FUNCTION_BLOCK "State_Machine2"   // FB71, GRAPH
VERSION : 0.1
// stored: AcknowledgeErrorsRequired true, AutoNumber false, GraphVersion 6.0, InitialValuesAcquisition false, IsIECCheckEnabled false, LanguageInNetworks LAD, LockOperatingMode false, PermanentILProcessingInMANMode false, SetENOAutomatically false, SkipSteps false, UDAEnableTagReadback false, WithAlarmHandling true
   // inherited from GRAPH_BASE
   VAR
      OFF_SQ_BASE : Bool;
   END_VAR
   VAR_INPUT
      OFF_SQ { ExternalAccessible := 'False'; ExternalVisible := 'False'; ExternalWritable := 'False'} : Bool := false;   // Disattiva catena / Turn sequence off
      INIT_SQ { ExternalAccessible := 'False'; ExternalVisible := 'False'; ExternalWritable := 'False'} : Bool := false;   // Imposta catena nello stato iniziale / Set sequence to initial state
      ACK_EF { ExternalAccessible := 'False'; ExternalVisible := 'False'; ExternalWritable := 'False'} : Bool := false;   // Conferma tutti gli errori e le anomalie / Acknowledge all errors and faults
      S_PREV { ExternalAccessible := 'False'; ExternalVisible := 'False'; ExternalWritable := 'False'} : Bool := false;   // Emetti il passo precedente nel parametro S_NO / Output previous step in parameter S_NO
      S_NEXT { ExternalAccessible := 'False'; ExternalVisible := 'False'; ExternalWritable := 'False'} : Bool := false;   // Visualizza passo successivo nel parametro S_NO / Indicate next step in parameter S_NO
      SW_AUTO { ExternalAccessible := 'False'; ExternalVisible := 'False'; ExternalWritable := 'False'} : Bool := false;   // Imposta funzionamento automatico / Automatic mode
      SW_TAP { ExternalAccessible := 'False'; ExternalVisible := 'False'; ExternalWritable := 'False'} : Bool := false;   // Semiautomatico/Avanza con transizione / Semiautomatic/switch with transition
      SW_TOP { ExternalAccessible := 'False'; ExternalVisible := 'False'; ExternalWritable := 'False'} : Bool := false;   // Semiautomatico/Ignora transizione / Semiautomatic/ignore transition
      SW_MAN { ExternalAccessible := 'False'; ExternalVisible := 'False'; ExternalWritable := 'False'} : Bool := false;   // Funzionamento manuale / Manual mode
      S_SEL { ExternalAccessible := 'False'; ExternalVisible := 'False'; ExternalWritable := 'False'} : Int := 0;   // Seleziona passo da visualizzare in S_NO / Select step to be output to S_NO
      S_ON { ExternalAccessible := 'False'; ExternalVisible := 'False'; ExternalWritable := 'False'} : Bool := false;   // Attiva passo visualizzato nel parametro S_NO / Activate step indicated in S_NO
      S_OFF { ExternalAccessible := 'False'; ExternalVisible := 'False'; ExternalWritable := 'False'} : Bool := false;   // Disattiva passo visualizzato nel parametro S_NO / Deactivate step indicated S_NO
      T_PUSH { ExternalAccessible := 'False'; ExternalVisible := 'False'; ExternalWritable := 'False'} : Bool := false;   // Abilita commutazione per la transizione nel funzionamento semiautomatico / Enable transition to switch in semi automatic mode
   END_VAR
   VAR_OUTPUT
      S_NO { ExternalAccessible := 'False'; ExternalVisible := 'False'; ExternalWritable := 'False'} : Int := 0;   // Numero del passo / Step number
      S_MORE { ExternalAccessible := 'False'; ExternalVisible := 'False'; ExternalWritable := 'False'} : Bool := false;   // Sono presenti altri passi e possono essere visualizzati in S_NO. / More steps are available and can be shown in S_NO
      S_ACTIVE { ExternalAccessible := 'False'; ExternalVisible := 'False'; ExternalWritable := 'False'} : Bool := false;   // Il passo visualizzato nel parametro S_NO è attivo / Step indicated in S_NO is active
      ERR_FLT { ExternalAccessible := 'False'; ExternalVisible := 'False'; ExternalWritable := 'False'} : Bool := false;   // Errore cumulativo interlock o supervisione / Interlock or supervision group error
      AUTO_ON { ExternalAccessible := 'False'; ExternalVisible := 'False'; ExternalWritable := 'False'} : Bool := false;   // Funzionamento automatico attivo / Automatic mode is active
      TAP_ON { ExternalAccessible := 'False'; ExternalVisible := 'False'; ExternalWritable := 'False'} : Bool := false;   // Funzionamento semiautomatico/Passo con transizione attivo / Semiautomatic mode/step with transition enabled
      TOP_ON { ExternalAccessible := 'False'; ExternalVisible := 'False'; ExternalWritable := 'False'} : Bool := false;   // Semiautomatico/Ignora transizione attivo / Semiautomatic mode/ignore transition enabled
      MAN_ON { ExternalAccessible := 'False'; ExternalVisible := 'False'; ExternalWritable := 'False'} : Bool := false;   // Funzionamento manuale attivo / Manual mode is active
   END_VAR
BEGIN
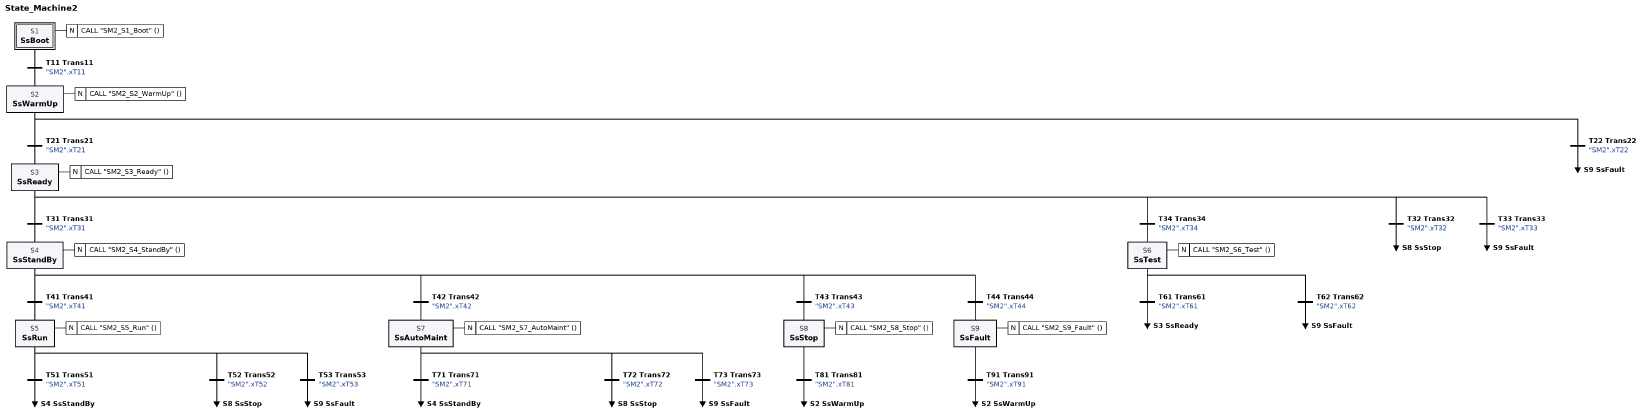
   // sequencer 1: State Machine Battery
   INITIAL_STEP SsBoot:   // S1, max time T#10S, warning time T#7S
              N    CALL "SM2_S1_Boot" ()
   END_STEP
   TRANSITION Trans11 FROM SsBoot TO SsWarmUp   // T11
      := "SM2".xT11;
   END_TRANSITION
   STEP SsWarmUp:   // S2, max time T#10S, warning time T#7S
              N    CALL "SM2_S2_WarmUp" ()
   END_STEP
   TRANSITION Trans21 FROM SsWarmUp TO SsReady   // T21
      := "SM2".xT21;
   END_TRANSITION
   TRANSITION Trans22 FROM SsWarmUp TO SsFault   // T22, jump
      := "SM2".xT22;
   END_TRANSITION
   STEP SsReady:   // S3, max time T#10S, warning time T#7S
              N    CALL "SM2_S3_Ready" ()
   END_STEP
   TRANSITION Trans31 FROM SsReady TO SsStandBy   // T31
      := "SM2".xT31;
   END_TRANSITION
   TRANSITION Trans34 FROM SsReady TO SsTest   // T34
      := "SM2".xT34;
   END_TRANSITION
   TRANSITION Trans32 FROM SsReady TO SsStop   // T32, jump
      := "SM2".xT32;
   END_TRANSITION
   TRANSITION Trans33 FROM SsReady TO SsFault   // T33, jump
      := "SM2".xT33;
   END_TRANSITION
   STEP SsStandBy:   // S4, max time T#10S, warning time T#7S
              N    CALL "SM2_S4_StandBy" ()
   END_STEP
   TRANSITION Trans41 FROM SsStandBy TO SsRun   // T41
      := "SM2".xT41;
   END_TRANSITION
   TRANSITION Trans42 FROM SsStandBy TO SsAutoMaint   // T42
      := "SM2".xT42;
   END_TRANSITION
   TRANSITION Trans43 FROM SsStandBy TO SsStop   // T43
      := "SM2".xT43;
   END_TRANSITION
   TRANSITION Trans44 FROM SsStandBy TO SsFault   // T44
      := "SM2".xT44;
   END_TRANSITION
   STEP SsRun:   // S5, max time T#10S, warning time T#7S
              N    CALL "SM2_S5_Run" ()
   END_STEP
   TRANSITION Trans51 FROM SsRun TO SsStandBy   // T51, jump
      := "SM2".xT51;
   END_TRANSITION
   TRANSITION Trans52 FROM SsRun TO SsStop   // T52, jump
      := "SM2".xT52;
   END_TRANSITION
   TRANSITION Trans53 FROM SsRun TO SsFault   // T53, jump
      := "SM2".xT53;
   END_TRANSITION
   STEP SsTest:   // S6, max time T#10S, warning time T#7S
              N    CALL "SM2_S6_Test" ()
   END_STEP
   TRANSITION Trans61 FROM SsTest TO SsReady   // T61, jump
      := "SM2".xT61;
   END_TRANSITION
   TRANSITION Trans62 FROM SsTest TO SsFault   // T62, jump
      := "SM2".xT62;
   END_TRANSITION
   STEP SsAutoMaint:   // S7, max time T#10S, warning time T#7S
              N    CALL "SM2_S7_AutoMaint" ()
   END_STEP
   TRANSITION Trans71 FROM SsAutoMaint TO SsStandBy   // T71, jump
      := "SM2".xT71;
   END_TRANSITION
   TRANSITION Trans72 FROM SsAutoMaint TO SsStop   // T72, jump
      := "SM2".xT72;
   END_TRANSITION
   TRANSITION Trans73 FROM SsAutoMaint TO SsFault   // T73, jump
      := "SM2".xT73;
   END_TRANSITION
   STEP SsStop:   // S8, max time T#10S, warning time T#7S
              N    CALL "SM2_S8_Stop" ()
   END_STEP
   TRANSITION Trans81 FROM SsStop TO SsWarmUp   // T81, jump
      := "SM2".xT81;
   END_TRANSITION
   STEP SsFault:   // S9, max time T#10S, warning time T#7S
              N    CALL "SM2_S9_Fault" ()
   END_STEP
   TRANSITION Trans91 FROM SsFault TO SsWarmUp   // T91, jump
      := "SM2".xT91;
   END_TRANSITION
END_FUNCTION_BLOCK

FUNCTION "LOGIC_PE_1" : Void   // FC7, LAD
{ S7_Optimized_Access := 'TRUE' }
VERSION : 0.1
// stored: AutoNumber true, IsIECCheckEnabled false, SetENOAutomatically false, UDAEnableTagReadback false
   VAR_TEMP
      rVac : Real;
   END_VAR
   VAR_TEMP   // added for the SCL form of the ladder/FBD networks
      _w1 : Bool;
      _w2 : Bool;
      _w3 : Bool;
   END_VAR
BEGIN

REGION Network 1: Write value of Password, P mode and Q mode - to check
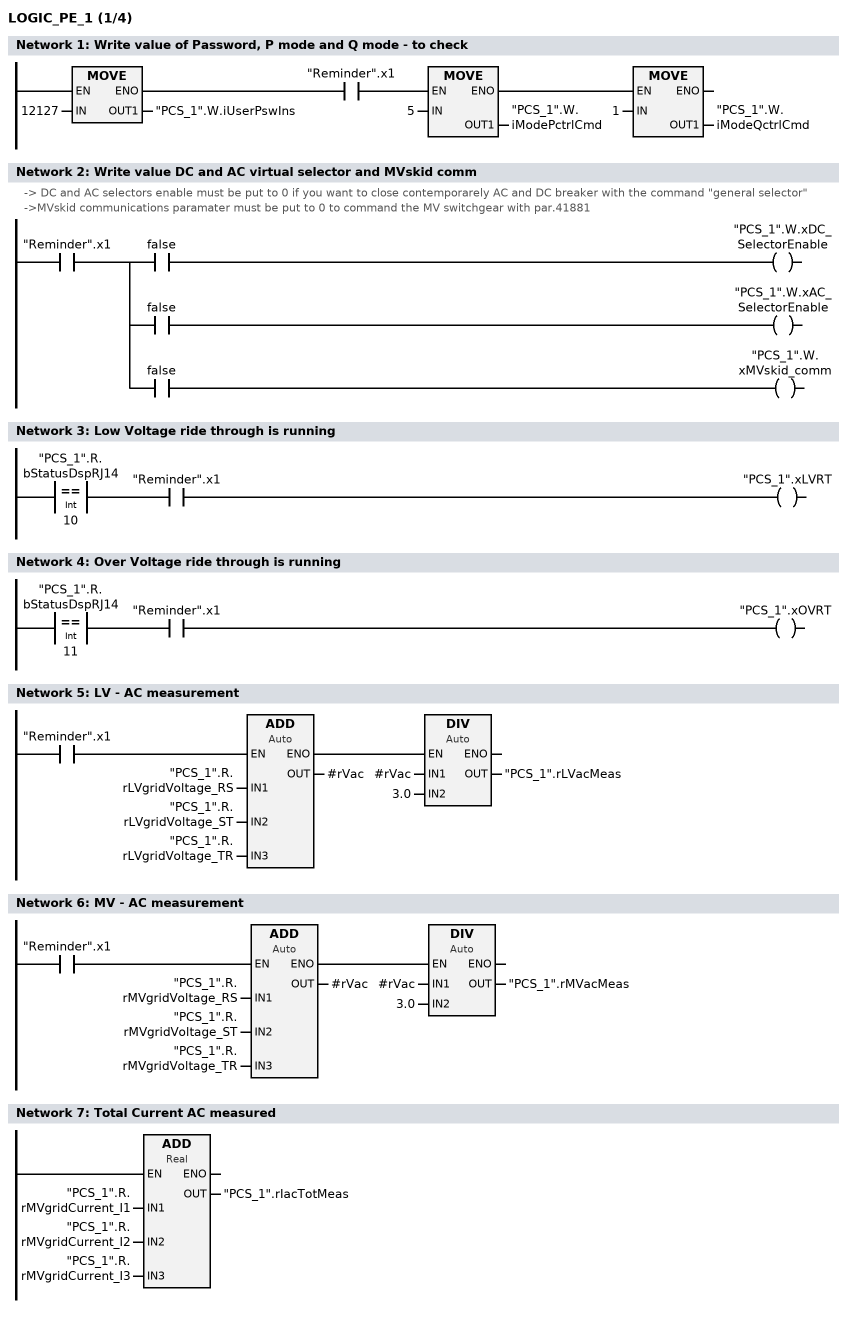
   RUNG wire#powerrail
      Move(in := 12127, out1 => "PCS_1".W.iUserPswIns)
      Contact( "Reminder".x1 )
      Move(in := 5, out1 => "PCS_1".W.iModePctrlCmd)
      Move(in := 1, out1 => "PCS_1".W.iModeQctrlCmd)
   END_RUNG
   // the same network as SCL:
   "PCS_1".W.iUserPswIns := 12127;
   IF "Reminder".x1 THEN
       "PCS_1".W.iModePctrlCmd := 5;
       "PCS_1".W.iModeQctrlCmd := 1;
   END_IF;
END_REGION

REGION Network 2: Write value DC and AC virtual selector and MVskid comm
   // -> DC and AC selectors enable must be put to 0 if you want to close contemporarely AC and DC breaker with the command "general selector"
   // ->MVskid communications paramater must be put to 0 to command the MV switchgear with par.41881
   RUNG wire#powerrail
      Contact( "Reminder".x1 )
      wire#w1
      Contact( false )
      Coil( "PCS_1".W.xDC_SelectorEnable )
   END_RUNG
   RUNG wire#w1
      Contact( false )
      Coil( "PCS_1".W.xAC_SelectorEnable )
   END_RUNG
   RUNG wire#w1
      Contact( false )
      Coil( "PCS_1".W.xMVskid_comm )
   END_RUNG
   // the same network as SCL:
   "PCS_1".W.xDC_SelectorEnable := "Reminder".x1 AND false;
   "PCS_1".W.xAC_SelectorEnable := "Reminder".x1 AND false;
   "PCS_1".W.xMVskid_comm := "Reminder".x1 AND false;
END_REGION

REGION Network 3: Low Voltage ride through is running
   RUNG wire#powerrail
      { S7_Templates := "SrcType := Int" } EQ_Contact(in1 := "PCS_1".R.bStatusDspRJ14, in2 := 10)
      Contact( "Reminder".x1 )
      Coil( "PCS_1".xLVRT )
   END_RUNG
   // the same network as SCL:
   "PCS_1".xLVRT := ("PCS_1".R.bStatusDspRJ14 = 10) AND "Reminder".x1;
END_REGION

REGION Network 4: Over Voltage ride through is running
   RUNG wire#powerrail
      { S7_Templates := "SrcType := Int" } EQ_Contact(in1 := "PCS_1".R.bStatusDspRJ14, in2 := 11)
      Contact( "Reminder".x1 )
      Coil( "PCS_1".xOVRT )
   END_RUNG
   // the same network as SCL:
   "PCS_1".xOVRT := ("PCS_1".R.bStatusDspRJ14 = 11) AND "Reminder".x1;
END_REGION

REGION Network 5: LV - AC measurement
   RUNG wire#powerrail
      Contact( "Reminder".x1 )
      Add(in1 := "PCS_1".R.rLVgridVoltage_RS, in2 := "PCS_1".R.rLVgridVoltage_ST, in3 := "PCS_1".R.rLVgridVoltage_TR, out => #rVac)
      Div(in1 := #rVac, in2 := 3.0, out => "PCS_1".rLVacMeas)
   END_RUNG
   // the same network as SCL:
   IF "Reminder".x1 THEN
       #rVac := "PCS_1".R.rLVgridVoltage_RS + "PCS_1".R.rLVgridVoltage_ST + "PCS_1".R.rLVgridVoltage_TR;
       "PCS_1".rLVacMeas := #rVac / 3.0;
   END_IF;
END_REGION

REGION Network 6: MV - AC measurement
   RUNG wire#powerrail
      Contact( "Reminder".x1 )
      Add(in1 := "PCS_1".R.rMVgridVoltage_RS, in2 := "PCS_1".R.rMVgridVoltage_ST, in3 := "PCS_1".R.rMVgridVoltage_TR, out => #rVac)
      Div(in1 := #rVac, in2 := 3.0, out => "PCS_1".rMVacMeas)
   END_RUNG
   // the same network as SCL:
   IF "Reminder".x1 THEN
       #rVac := "PCS_1".R.rMVgridVoltage_RS + "PCS_1".R.rMVgridVoltage_ST + "PCS_1".R.rMVgridVoltage_TR;
       "PCS_1".rMVacMeas := #rVac / 3.0;
   END_IF;
END_REGION

REGION Network 7: Total Current AC measured
   RUNG wire#powerrail
      { S7_Templates := "SrcType := Real" } Add(in1 := "PCS_1".R.rMVgridCurrent_I1, in2 := "PCS_1".R.rMVgridCurrent_I2, in3 := "PCS_1".R.rMVgridCurrent_I3, out => "PCS_1".rIacTotMeas)
   END_RUNG
   // the same network as SCL:
   "PCS_1".rIacTotMeas := "PCS_1".R.rMVgridCurrent_I1 + "PCS_1".R.rMVgridCurrent_I2 + "PCS_1".R.rMVgridCurrent_I3;
END_REGION

REGION Network 8: Inverter status
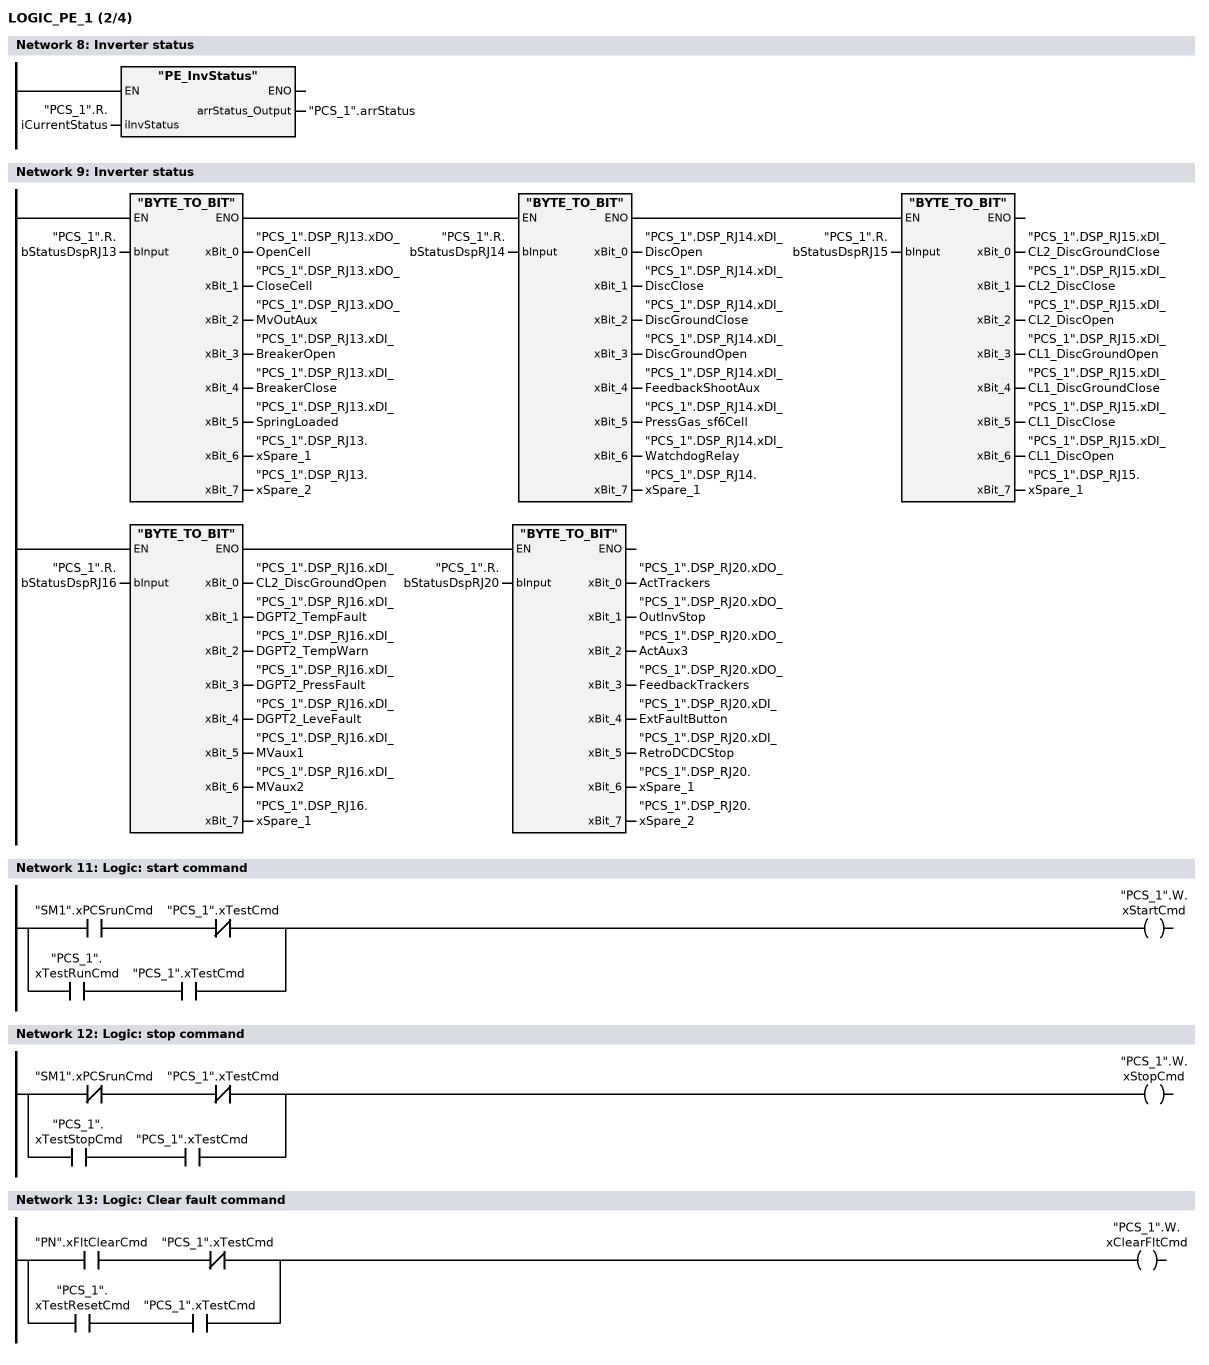
   RUNG wire#powerrail
      "PE_InvStatus"(iInvStatus := "PCS_1".R.iCurrentStatus, arrStatus_Output => "PCS_1".arrStatus)
   END_RUNG
   // the same network as SCL:
   "PE_InvStatus"(iInvStatus := "PCS_1".R.iCurrentStatus, arrStatus_Output => "PCS_1".arrStatus);
END_REGION

REGION Network 9: Inverter status
   RUNG wire#powerrail
      "BYTE_TO_BIT"(bInput := "PCS_1".R.bStatusDspRJ13, xBit_0 => "PCS_1".DSP_RJ13.xDO_OpenCell, xBit_1 => "PCS_1".DSP_RJ13.xDO_CloseCell, xBit_2 => "PCS_1".DSP_RJ13.xDO_MvOutAux, xBit_3 => "PCS_1".DSP_RJ13.xDI_BreakerOpen, xBit_4 => "PCS_1".DSP_RJ13.xDI_BreakerClose, xBit_5 => "PCS_1".DSP_RJ13.xDI_SpringLoaded, xBit_6 => "PCS_1".DSP_RJ13.xSpare_1, xBit_7 => "PCS_1".DSP_RJ13.xSpare_2)
      "BYTE_TO_BIT"(bInput := "PCS_1".R.bStatusDspRJ14, xBit_0 => "PCS_1".DSP_RJ14.xDI_DiscOpen, xBit_1 => "PCS_1".DSP_RJ14.xDI_DiscClose, xBit_2 => "PCS_1".DSP_RJ14.xDI_DiscGroundClose, xBit_3 => "PCS_1".DSP_RJ14.xDI_DiscGroundOpen, xBit_4 => "PCS_1".DSP_RJ14.xDI_FeedbackShootAux, xBit_5 => "PCS_1".DSP_RJ14.xDI_PressGas_sf6Cell, xBit_6 => "PCS_1".DSP_RJ14.xDI_WatchdogRelay, xBit_7 => "PCS_1".DSP_RJ14.xSpare_1)
      "BYTE_TO_BIT"(bInput := "PCS_1".R.bStatusDspRJ15, xBit_0 => "PCS_1".DSP_RJ15.xDI_CL2_DiscGroundClose, xBit_1 => "PCS_1".DSP_RJ15.xDI_CL2_DiscClose, xBit_2 => "PCS_1".DSP_RJ15.xDI_CL2_DiscOpen, xBit_3 => "PCS_1".DSP_RJ15.xDI_CL1_DiscGroundOpen, xBit_4 => "PCS_1".DSP_RJ15.xDI_CL1_DiscGroundClose, xBit_5 => "PCS_1".DSP_RJ15.xDI_CL1_DiscClose, xBit_6 => "PCS_1".DSP_RJ15.xDI_CL1_DiscOpen, xBit_7 => "PCS_1".DSP_RJ15.xSpare_1)
   END_RUNG
   RUNG wire#powerrail
      "BYTE_TO_BIT"(bInput := "PCS_1".R.bStatusDspRJ16, xBit_0 => "PCS_1".DSP_RJ16.xDI_CL2_DiscGroundOpen, xBit_1 => "PCS_1".DSP_RJ16.xDI_DGPT2_TempFault, xBit_2 => "PCS_1".DSP_RJ16.xDI_DGPT2_TempWarn, xBit_3 => "PCS_1".DSP_RJ16.xDI_DGPT2_PressFault, xBit_4 => "PCS_1".DSP_RJ16.xDI_DGPT2_LeveFault, xBit_5 => "PCS_1".DSP_RJ16.xDI_MVaux1, xBit_6 => "PCS_1".DSP_RJ16.xDI_MVaux2, xBit_7 => "PCS_1".DSP_RJ16.xSpare_1)
      "BYTE_TO_BIT"(bInput := "PCS_1".R.bStatusDspRJ20, xBit_0 => "PCS_1".DSP_RJ20.xDO_ActTrackers, xBit_1 => "PCS_1".DSP_RJ20.xDO_OutInvStop, xBit_2 => "PCS_1".DSP_RJ20.xDO_ActAux3, xBit_3 => "PCS_1".DSP_RJ20.xDO_FeedbackTrackers, xBit_4 => "PCS_1".DSP_RJ20.xDI_ExtFaultButton, xBit_5 => "PCS_1".DSP_RJ20.xDI_RetroDCDCStop, xBit_6 => "PCS_1".DSP_RJ20.xSpare_1, xBit_7 => "PCS_1".DSP_RJ20.xSpare_2)
   END_RUNG
   // the same network as SCL:
   "BYTE_TO_BIT"(bInput := "PCS_1".R.bStatusDspRJ13,
                 xBit_0 => "PCS_1".DSP_RJ13.xDO_OpenCell,
                 xBit_1 => "PCS_1".DSP_RJ13.xDO_CloseCell,
                 xBit_2 => "PCS_1".DSP_RJ13.xDO_MvOutAux,
                 xBit_3 => "PCS_1".DSP_RJ13.xDI_BreakerOpen,
                 xBit_4 => "PCS_1".DSP_RJ13.xDI_BreakerClose,
                 xBit_5 => "PCS_1".DSP_RJ13.xDI_SpringLoaded,
                 xBit_6 => "PCS_1".DSP_RJ13.xSpare_1,
                 xBit_7 => "PCS_1".DSP_RJ13.xSpare_2,
                 ENO => #_w1);
   "BYTE_TO_BIT"(EN := #_w1,
                 bInput := "PCS_1".R.bStatusDspRJ14,
                 xBit_0 => "PCS_1".DSP_RJ14.xDI_DiscOpen,
                 xBit_1 => "PCS_1".DSP_RJ14.xDI_DiscClose,
                 xBit_2 => "PCS_1".DSP_RJ14.xDI_DiscGroundClose,
                 xBit_3 => "PCS_1".DSP_RJ14.xDI_DiscGroundOpen,
                 xBit_4 => "PCS_1".DSP_RJ14.xDI_FeedbackShootAux,
                 xBit_5 => "PCS_1".DSP_RJ14.xDI_PressGas_sf6Cell,
                 xBit_6 => "PCS_1".DSP_RJ14.xDI_WatchdogRelay,
                 xBit_7 => "PCS_1".DSP_RJ14.xSpare_1,
                 ENO => #_w2);
   IF #_w2 THEN
       "BYTE_TO_BIT"(bInput := "PCS_1".R.bStatusDspRJ15,
                     xBit_0 => "PCS_1".DSP_RJ15.xDI_CL2_DiscGroundClose,
                     xBit_1 => "PCS_1".DSP_RJ15.xDI_CL2_DiscClose,
                     xBit_2 => "PCS_1".DSP_RJ15.xDI_CL2_DiscOpen,
                     xBit_3 => "PCS_1".DSP_RJ15.xDI_CL1_DiscGroundOpen,
                     xBit_4 => "PCS_1".DSP_RJ15.xDI_CL1_DiscGroundClose,
                     xBit_5 => "PCS_1".DSP_RJ15.xDI_CL1_DiscClose,
                     xBit_6 => "PCS_1".DSP_RJ15.xDI_CL1_DiscOpen,
                     xBit_7 => "PCS_1".DSP_RJ15.xSpare_1);
   END_IF;
   "BYTE_TO_BIT"(bInput := "PCS_1".R.bStatusDspRJ16,
                 xBit_0 => "PCS_1".DSP_RJ16.xDI_CL2_DiscGroundOpen,
                 xBit_1 => "PCS_1".DSP_RJ16.xDI_DGPT2_TempFault,
                 xBit_2 => "PCS_1".DSP_RJ16.xDI_DGPT2_TempWarn,
                 xBit_3 => "PCS_1".DSP_RJ16.xDI_DGPT2_PressFault,
                 xBit_4 => "PCS_1".DSP_RJ16.xDI_DGPT2_LeveFault,
                 xBit_5 => "PCS_1".DSP_RJ16.xDI_MVaux1,
                 xBit_6 => "PCS_1".DSP_RJ16.xDI_MVaux2,
                 xBit_7 => "PCS_1".DSP_RJ16.xSpare_1,
                 ENO => #_w3);
   IF #_w3 THEN
       "BYTE_TO_BIT"(bInput := "PCS_1".R.bStatusDspRJ20,
                     xBit_0 => "PCS_1".DSP_RJ20.xDO_ActTrackers,
                     xBit_1 => "PCS_1".DSP_RJ20.xDO_OutInvStop,
                     xBit_2 => "PCS_1".DSP_RJ20.xDO_ActAux3,
                     xBit_3 => "PCS_1".DSP_RJ20.xDO_FeedbackTrackers,
                     xBit_4 => "PCS_1".DSP_RJ20.xDI_ExtFaultButton,
                     xBit_5 => "PCS_1".DSP_RJ20.xDI_RetroDCDCStop,
                     xBit_6 => "PCS_1".DSP_RJ20.xSpare_1,
                     xBit_7 => "PCS_1".DSP_RJ20.xSpare_2);
   END_IF;
END_REGION

REGION Network 11: Logic: start command
   RUNG wire#powerrail
      Contact( "SM1".xPCSrunCmd )
      I_Contact( "PCS_1".xTestCmd )
      wire#w1
      Coil( "PCS_1".W.xStartCmd )
   END_RUNG
   RUNG wire#powerrail
      Contact( "PCS_1".xTestRunCmd )
      Contact( "PCS_1".xTestCmd )
   END_RUNG wire#w1
   // the same network as SCL:
   "PCS_1".W.xStartCmd := ("SM1".xPCSrunCmd AND NOT "PCS_1".xTestCmd) OR ("PCS_1".xTestRunCmd AND "PCS_1".xTestCmd);
END_REGION

REGION Network 12: Logic: stop command
   RUNG wire#powerrail
      I_Contact( "SM1".xPCSrunCmd )
      I_Contact( "PCS_1".xTestCmd )
      wire#w1
      Coil( "PCS_1".W.xStopCmd )
   END_RUNG
   RUNG wire#powerrail
      Contact( "PCS_1".xTestStopCmd )
      Contact( "PCS_1".xTestCmd )
   END_RUNG wire#w1
   // the same network as SCL:
   "PCS_1".W.xStopCmd := (NOT "SM1".xPCSrunCmd AND NOT "PCS_1".xTestCmd) OR ("PCS_1".xTestStopCmd AND "PCS_1".xTestCmd);
END_REGION

REGION Network 13: Logic: Clear fault command
   RUNG wire#powerrail
      Contact( "PN".xFltClearCmd )
      I_Contact( "PCS_1".xTestCmd )
      wire#w1
      Coil( "PCS_1".W.xClearFltCmd )
   END_RUNG
   RUNG wire#powerrail
      Contact( "PCS_1".xTestResetCmd )
      Contact( "PCS_1".xTestCmd )
   END_RUNG wire#w1
   // the same network as SCL:
   "PCS_1".W.xClearFltCmd := ("PN".xFltClearCmd AND NOT "PCS_1".xTestCmd) OR ("PCS_1".xTestResetCmd AND "PCS_1".xTestCmd);
END_REGION

REGION Network 14: Logic : PPC enable command
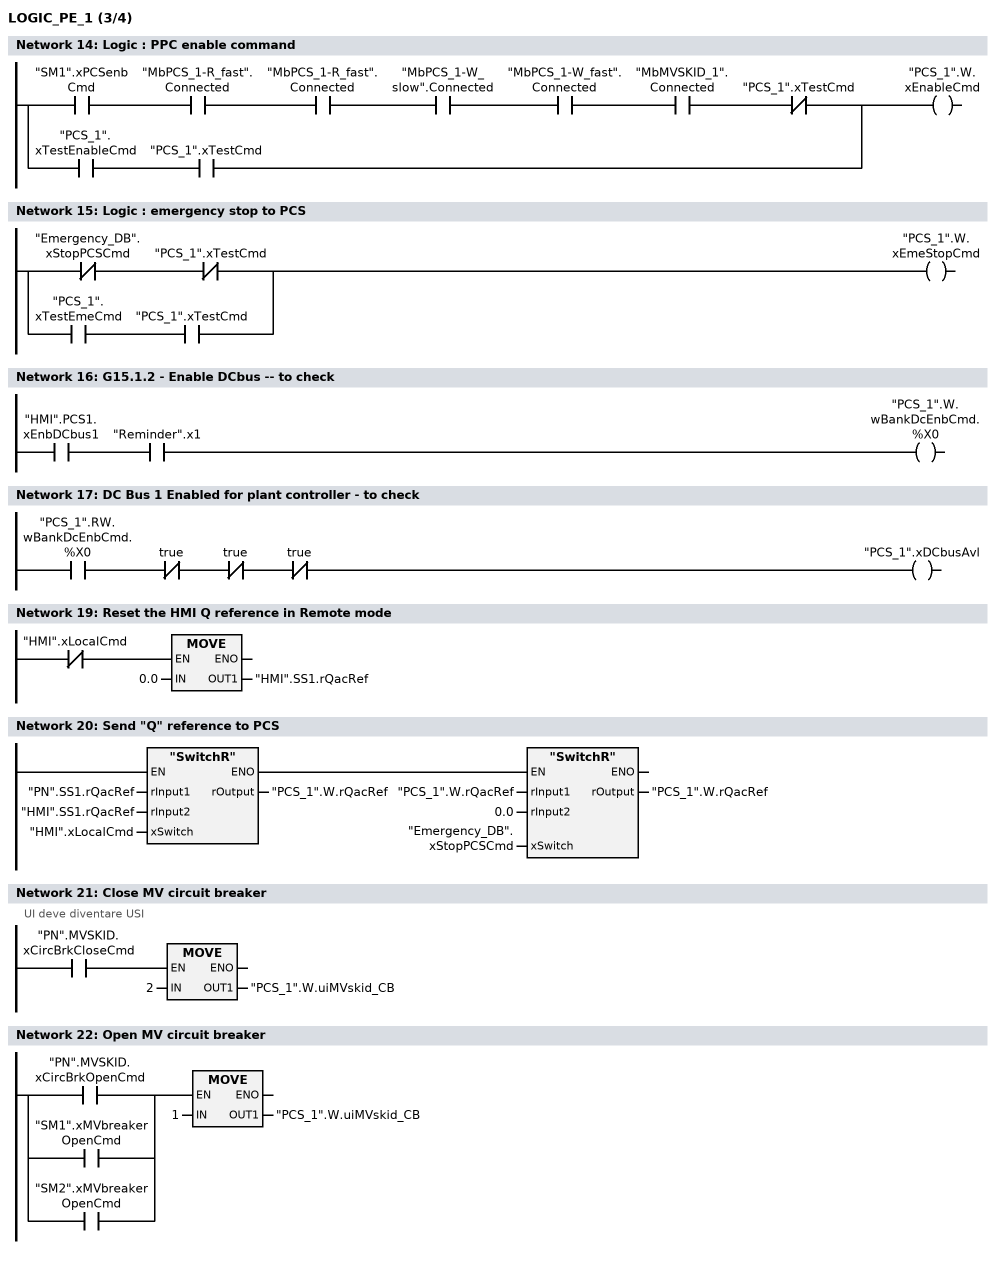
   RUNG wire#powerrail
      Contact( "SM1".xPCSenbCmd )
      Contact( "MbPCS_1-R_fast".Connected )
      Contact( "MbPCS_1-R_fast".Connected )
      Contact( "MbPCS_1-W_slow".Connected )
      Contact( "MbPCS_1-W_fast".Connected )
      Contact( "MbMVSKID_1".Connected )
      I_Contact( "PCS_1".xTestCmd )
      wire#w1
      Coil( "PCS_1".W.xEnableCmd )
   END_RUNG
   RUNG wire#powerrail
      Contact( "PCS_1".xTestEnableCmd )
      Contact( "PCS_1".xTestCmd )
   END_RUNG wire#w1
   // the same network as SCL:
   "PCS_1".W.xEnableCmd := ("SM1".xPCSenbCmd AND "MbPCS_1-R_fast".Connected AND "MbPCS_1-R_fast".Connected AND "MbPCS_1-W_slow".Connected AND "MbPCS_1-W_fast".Connected AND "MbMVSKID_1".Connected AND NOT "PCS_1".xTestCmd) OR ("PCS_1".xTestEnableCmd AND "PCS_1".xTestCmd);
END_REGION

REGION Network 15: Logic : emergency stop to PCS
   RUNG wire#powerrail
      I_Contact( "Emergency_DB".xStopPCSCmd )
      I_Contact( "PCS_1".xTestCmd )
      wire#w1
      Coil( "PCS_1".W.xEmeStopCmd )
   END_RUNG
   RUNG wire#powerrail
      Contact( "PCS_1".xTestEmeCmd )
      Contact( "PCS_1".xTestCmd )
   END_RUNG wire#w1
   // the same network as SCL:
   "PCS_1".W.xEmeStopCmd := (NOT "Emergency_DB".xStopPCSCmd AND NOT "PCS_1".xTestCmd) OR ("PCS_1".xTestEmeCmd AND "PCS_1".xTestCmd);
END_REGION

REGION Network 16: G15.1.2 - Enable DCbus -- to check
   RUNG wire#powerrail
      Contact( "HMI".PCS1.xEnbDCbus1 )
      Contact( "Reminder".x1 )
      Coil( "PCS_1".W.wBankDcEnbCmd.%X0 )
   END_RUNG
   // the same network as SCL:
   "PCS_1".W.wBankDcEnbCmd.%X0 := "HMI".PCS1.xEnbDCbus1 AND "Reminder".x1;
END_REGION

REGION Network 17: DC Bus 1 Enabled for plant controller - to check
   RUNG wire#powerrail
      Contact( "PCS_1".RW.wBankDcEnbCmd.%X0 )
      I_Contact( true )
      I_Contact( true )
      I_Contact( true )
      Coil( "PCS_1".xDCbusAvl )
   END_RUNG
   // the same network as SCL:
   "PCS_1".xDCbusAvl := "PCS_1".RW.wBankDcEnbCmd.%X0 AND NOT true AND NOT true AND NOT true;
END_REGION

REGION Network 19: Reset the HMI Q reference in Remote mode
   RUNG wire#powerrail
      I_Contact( "HMI".xLocalCmd )
      Move(in := 0.0, out1 => "HMI".SS1.rQacRef)
   END_RUNG
   // the same network as SCL:
   IF NOT "HMI".xLocalCmd THEN "HMI".SS1.rQacRef := 0.0; END_IF;
END_REGION

REGION Network 20: Send "Q" reference to PCS
   RUNG wire#powerrail
      "SwitchR"(rInput1 := "PN".SS1.rQacRef, rInput2 := "HMI".SS1.rQacRef, xSwitch := "HMI".xLocalCmd, rOutput => "PCS_1".W.rQacRef)
      "SwitchR"(rInput1 := "PCS_1".W.rQacRef, rInput2 := 0.0, xSwitch := "Emergency_DB".xStopPCSCmd, rOutput => "PCS_1".W.rQacRef)
   END_RUNG
   // the same network as SCL:
   "SwitchR"(rInput1 := "PN".SS1.rQacRef,
             rInput2 := "HMI".SS1.rQacRef,
             xSwitch := "HMI".xLocalCmd,
             rOutput => "PCS_1".W.rQacRef,
             ENO => #_w1);
   IF #_w1 THEN
       "SwitchR"(rInput1 := "PCS_1".W.rQacRef,
                 rInput2 := 0.0,
                 xSwitch := "Emergency_DB".xStopPCSCmd,
                 rOutput => "PCS_1".W.rQacRef);
   END_IF;
END_REGION

REGION Network 21: Close MV circuit breaker
   // UI deve diventare USI
   RUNG wire#powerrail
      Contact( "PN".MVSKID.xCircBrkCloseCmd )
      Move(in := 2, out1 => "PCS_1".W.uiMVskid_CB)
   END_RUNG
   // the same network as SCL:
   IF "PN".MVSKID.xCircBrkCloseCmd THEN "PCS_1".W.uiMVskid_CB := 2; END_IF;
END_REGION

REGION Network 22: Open MV circuit breaker
   RUNG wire#powerrail
      Contact( "PN".MVSKID.xCircBrkOpenCmd )
      wire#w1
      Move(in := 1, out1 => "PCS_1".W.uiMVskid_CB)
   END_RUNG
   RUNG wire#powerrail
      Contact( "SM1".xMVbreakerOpenCmd )
   END_RUNG wire#w1
   RUNG wire#powerrail
      Contact( "SM2".xMVbreakerOpenCmd )
   END_RUNG wire#w1
   // the same network as SCL:
   IF "PN".MVSKID.xCircBrkOpenCmd OR "SM1".xMVbreakerOpenCmd OR "SM2".xMVbreakerOpenCmd THEN
       "PCS_1".W.uiMVskid_CB := 1;
   END_IF;
END_REGION

REGION Network 23: MV SKID Fault
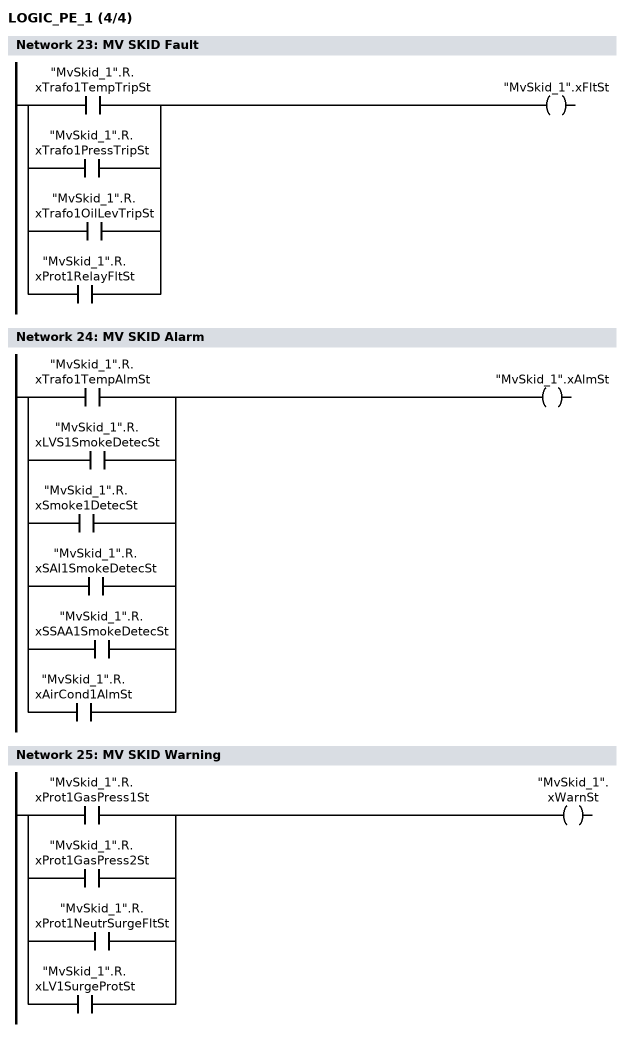
   RUNG wire#powerrail
      Contact( "MvSkid_1".R.xTrafo1TempTripSt )
      wire#w1
      Coil( "MvSkid_1".xFltSt )
   END_RUNG
   RUNG wire#powerrail
      Contact( "MvSkid_1".R.xTrafo1PressTripSt )
   END_RUNG wire#w1
   RUNG wire#powerrail
      Contact( "MvSkid_1".R.xTrafo1OilLevTripSt )
   END_RUNG wire#w1
   RUNG wire#powerrail
      Contact( "MvSkid_1".R.xProt1RelayFltSt )
   END_RUNG wire#w1
   // the same network as SCL:
   "MvSkid_1".xFltSt := "MvSkid_1".R.xTrafo1TempTripSt OR "MvSkid_1".R.xTrafo1PressTripSt OR "MvSkid_1".R.xTrafo1OilLevTripSt OR "MvSkid_1".R.xProt1RelayFltSt;
END_REGION

REGION Network 24: MV SKID Alarm
   RUNG wire#powerrail
      Contact( "MvSkid_1".R.xTrafo1TempAlmSt )
      wire#w1
      Coil( "MvSkid_1".xAlmSt )
   END_RUNG
   RUNG wire#powerrail
      Contact( "MvSkid_1".R.xLVS1SmokeDetecSt )
   END_RUNG wire#w1
   RUNG wire#powerrail
      Contact( "MvSkid_1".R.xSmoke1DetecSt )
   END_RUNG wire#w1
   RUNG wire#powerrail
      Contact( "MvSkid_1".R.xSAI1SmokeDetecSt )
   END_RUNG wire#w1
   RUNG wire#powerrail
      Contact( "MvSkid_1".R.xSSAA1SmokeDetecSt )
   END_RUNG wire#w1
   RUNG wire#powerrail
      Contact( "MvSkid_1".R.xAirCond1AlmSt )
   END_RUNG wire#w1
   // the same network as SCL:
   "MvSkid_1".xAlmSt := "MvSkid_1".R.xTrafo1TempAlmSt OR "MvSkid_1".R.xLVS1SmokeDetecSt OR "MvSkid_1".R.xSmoke1DetecSt OR "MvSkid_1".R.xSAI1SmokeDetecSt OR "MvSkid_1".R.xSSAA1SmokeDetecSt OR "MvSkid_1".R.xAirCond1AlmSt;
END_REGION

REGION Network 25: MV SKID Warning
   RUNG wire#powerrail
      Contact( "MvSkid_1".R.xProt1GasPress1St )
      wire#w1
      Coil( "MvSkid_1".xWarnSt )
   END_RUNG
   RUNG wire#powerrail
      Contact( "MvSkid_1".R.xProt1GasPress2St )
   END_RUNG wire#w1
   RUNG wire#powerrail
      Contact( "MvSkid_1".R.xProt1NeutrSurgeFltSt )
   END_RUNG wire#w1
   RUNG wire#powerrail
      Contact( "MvSkid_1".R.xLV1SurgeProtSt )
   END_RUNG wire#w1
   // the same network as SCL:
   "MvSkid_1".xWarnSt := "MvSkid_1".R.xProt1GasPress1St OR "MvSkid_1".R.xProt1GasPress2St OR "MvSkid_1".R.xProt1NeutrSurgeFltSt OR "MvSkid_1".R.xLV1SurgeProtSt;
END_REGION

REGION Network 26 (SCL): MV SKID Line Disconnector & Breaker Status
   "MvSkid_1".wLine1DiscSt.%X0 := "MvSkid_1".R.xLine1DiscOpenSt;
   "MvSkid_1".wLine1DiscSt.%X1 := "MvSkid_1".R.xLine1DiscCloseSt;
   "MvSkid_1".wLine1DiscSt.%X2 := "MvSkid_1".R.xLine1GndCloseSt;

   "MvSkid_1".wLine2DiscSt.%X0 := "MvSkid_1".R.xLine2DiscOpenSt;
   "MvSkid_1".wLine2DiscSt.%X1 := "MvSkid_1".R.xLine2DiscCloseSt;
   "MvSkid_1".wLine2DiscSt.%X2 := "MvSkid_1".R.xLine2GndCloseSt;

   "MvSkid_1".wProt1DiscSt.%X0 := "MvSkid_1".R.xProt1DiscOpenSt;
   "MvSkid_1".wProt1DiscSt.%X1 := "MvSkid_1".R.xProt1DiscCloseSt;
   "MvSkid_1".wProt1DiscSt.%X2 := "MvSkid_1".R.xProt1GndCloseSt;

   "MvSkid_1".wProt1CircBrkSt.%X0 := "MvSkid_1".R.xProt1CircBrkOpenSt;
   "MvSkid_1".wProt1CircBrkSt.%X1 := "MvSkid_1".R.xProt1CircBrkCloseSt;
END_REGION
END_FUNCTION

FUNCTION "MV SKID (PE)_1" : Void   // FC45, LAD
TITLE = ModBus TCP for MVSKID Power Electronics
{ S7_Optimized_Access := 'TRUE' }
VERSION : 0.1
// stored: AutoNumber false, IsIECCheckEnabled false, SetENOAutomatically false, UDAEnableTagReadback false
   VAR_TEMP   // added for the SCL form of the ladder/FBD networks
      _w1 : Bool;
   END_VAR
BEGIN

REGION Network 1: Function Modbus Client
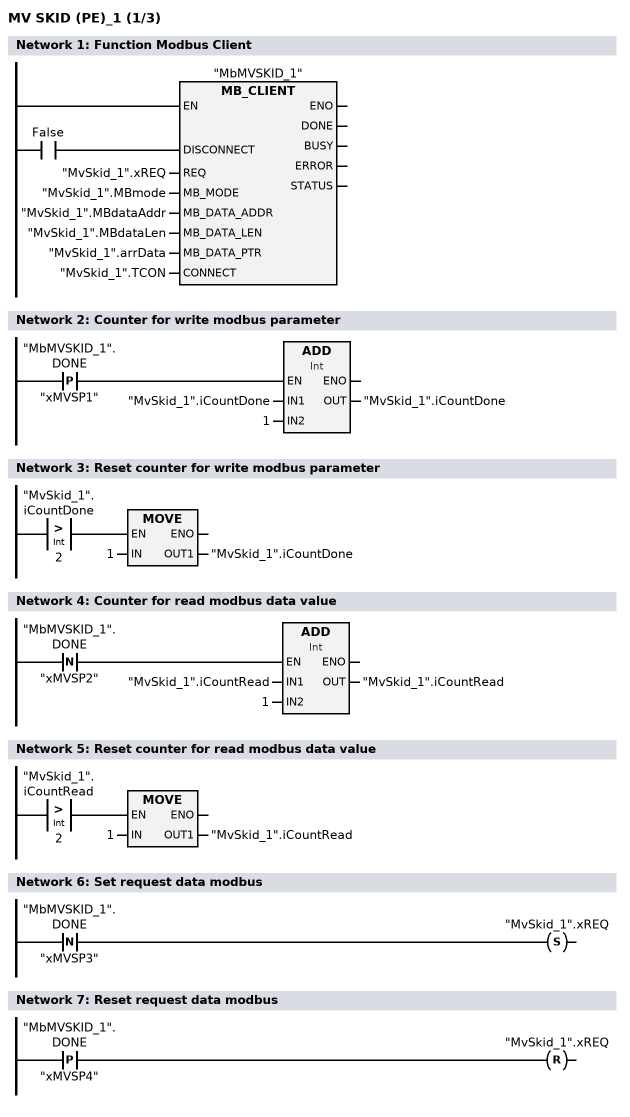
   RUNG wire#powerrail
      "MbMVSKID_1".MB_CLIENT(DISCONNECT := wire#w1, REQ := "MvSkid_1".xREQ, MB_MODE := "MvSkid_1".MBmode, MB_DATA_ADDR := "MvSkid_1".MBdataAddr, MB_DATA_LEN := "MvSkid_1".MBdataLen, MB_DATA_PTR := "MvSkid_1".arrData, CONNECT := "MvSkid_1".TCON, DONE =>, BUSY =>, ERROR =>, STATUS =>)
   END_RUNG
   RUNG wire#powerrail
      Contact( False )
   END_RUNG wire#w1
   // the same network as SCL:
   "MbMVSKID_1"(DISCONNECT := False,   // MB_CLIENT
                REQ := "MvSkid_1".xREQ,
                MB_MODE := "MvSkid_1".MBmode,
                MB_DATA_ADDR := "MvSkid_1".MBdataAddr,
                MB_DATA_LEN := "MvSkid_1".MBdataLen,
                MB_DATA_PTR := "MvSkid_1".arrData,
                CONNECT := "MvSkid_1".TCON);
END_REGION

REGION Network 2: Counter for write modbus parameter
   RUNG wire#powerrail
      P_Contact(operand := "MbMVSKID_1".DONE, bit := "xMVSP1")
      { S7_Templates := "SrcType := Int" } Add(in1 := "MvSkid_1".iCountDone, in2 := 1, out => "MvSkid_1".iCountDone)
   END_RUNG
   // the same network as SCL:
   #_w1 := "MbMVSKID_1".DONE AND NOT "xMVSP1";   // rising edge of "MbMVSKID_1".DONE
   "xMVSP1" := "MbMVSKID_1".DONE;
   IF #_w1 THEN "MvSkid_1".iCountDone := "MvSkid_1".iCountDone + 1; END_IF;
END_REGION

REGION Network 3: Reset counter for write modbus parameter
   RUNG wire#powerrail
      { S7_Templates := "SrcType := Int" } GT_Contact(in1 := "MvSkid_1".iCountDone, in2 := 2)
      Move(in := 1, out1 => "MvSkid_1".iCountDone)
   END_RUNG
   // the same network as SCL:
   IF "MvSkid_1".iCountDone > 2 THEN "MvSkid_1".iCountDone := 1; END_IF;
END_REGION

REGION Network 4: Counter for read modbus data value
   RUNG wire#powerrail
      N_Contact(operand := "MbMVSKID_1".DONE, bit := "xMVSP2")
      { S7_Templates := "SrcType := Int" } Add(in1 := "MvSkid_1".iCountRead, in2 := 1, out => "MvSkid_1".iCountRead)
   END_RUNG
   // the same network as SCL:
   #_w1 := NOT "MbMVSKID_1".DONE AND "xMVSP2";   // falling edge of "MbMVSKID_1".DONE
   "xMVSP2" := "MbMVSKID_1".DONE;
   IF #_w1 THEN "MvSkid_1".iCountRead := "MvSkid_1".iCountRead + 1; END_IF;
END_REGION

REGION Network 5: Reset counter for read modbus data value
   RUNG wire#powerrail
      { S7_Templates := "SrcType := Int" } GT_Contact(in1 := "MvSkid_1".iCountRead, in2 := 2)
      Move(in := 1, out1 => "MvSkid_1".iCountRead)
   END_RUNG
   // the same network as SCL:
   IF "MvSkid_1".iCountRead > 2 THEN "MvSkid_1".iCountRead := 1; END_IF;
END_REGION

REGION Network 6: Set request data modbus
   RUNG wire#powerrail
      N_Contact(operand := "MbMVSKID_1".DONE, bit := "xMVSP3")
      S_Coil( "MvSkid_1".xREQ )
   END_RUNG
   // the same network as SCL:
   #_w1 := NOT "MbMVSKID_1".DONE AND "xMVSP3";   // falling edge of "MbMVSKID_1".DONE
   "xMVSP3" := "MbMVSKID_1".DONE;
   IF #_w1 THEN "MvSkid_1".xREQ := TRUE; END_IF;
END_REGION

REGION Network 7: Reset request data modbus
   RUNG wire#powerrail
      P_Contact(operand := "MbMVSKID_1".DONE, bit := "xMVSP4")
      R_Coil( "MvSkid_1".xREQ )
   END_RUNG
   // the same network as SCL:
   #_w1 := "MbMVSKID_1".DONE AND NOT "xMVSP4";   // rising edge of "MbMVSKID_1".DONE
   "xMVSP4" := "MbMVSKID_1".DONE;
   IF #_w1 THEN "MvSkid_1".xREQ := FALSE; END_IF;
END_REGION

REGION Network 8: Write R_MVSKID parameter
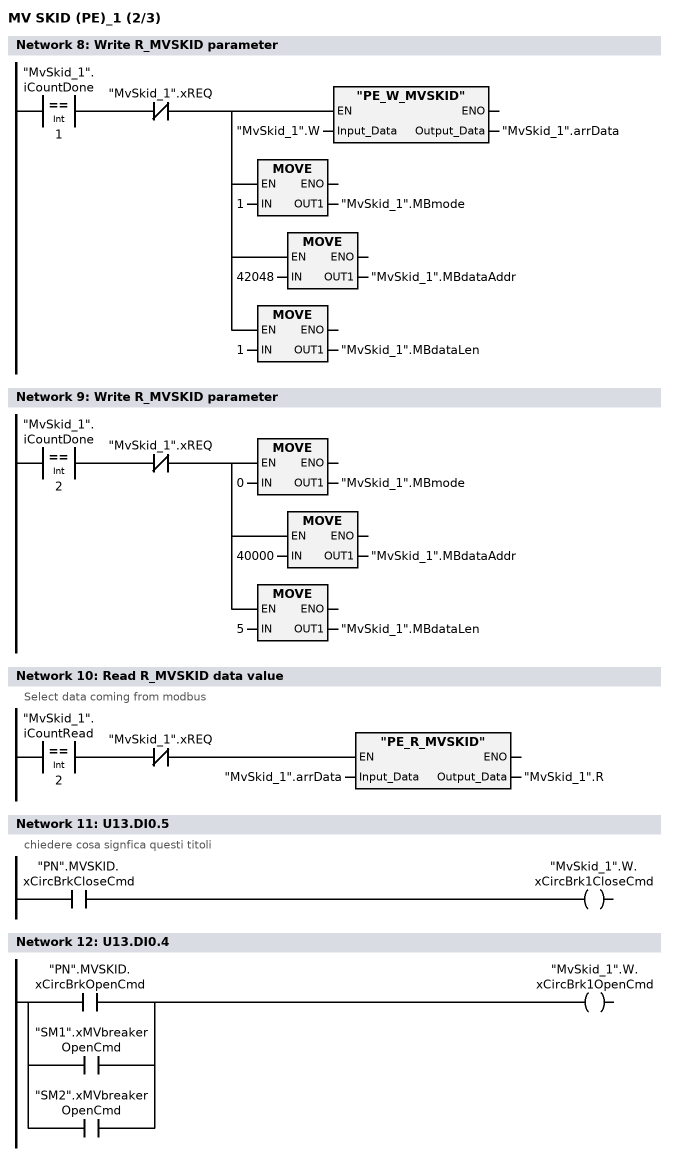
   RUNG wire#powerrail
      { S7_Templates := "SrcType := Int" } EQ_Contact(in1 := "MvSkid_1".iCountDone, in2 := 1)
      I_Contact( "MvSkid_1".xREQ )
      wire#w1
      "PE_W_MVSKID"(Input_Data := "MvSkid_1".W, Output_Data => "MvSkid_1".arrData)
   END_RUNG
   RUNG wire#w1
      Move(in := 1, out1 => "MvSkid_1".MBmode)
   END_RUNG
   RUNG wire#w1
      Move(in := 42048, out1 => "MvSkid_1".MBdataAddr)
   END_RUNG
   RUNG wire#w1
      Move(in := 1, out1 => "MvSkid_1".MBdataLen)
   END_RUNG
   // the same network as SCL:
   #_w1 := ("MvSkid_1".iCountDone = 1) AND NOT "MvSkid_1".xREQ;
   IF #_w1 THEN
       "PE_W_MVSKID"(Input_Data := "MvSkid_1".W, Output_Data => "MvSkid_1".arrData);
       "MvSkid_1".MBmode := 1;
       "MvSkid_1".MBdataAddr := 42048;
       "MvSkid_1".MBdataLen := 1;
   END_IF;
END_REGION

REGION Network 9: Write R_MVSKID parameter
   RUNG wire#powerrail
      { S7_Templates := "SrcType := Int" } EQ_Contact(in1 := "MvSkid_1".iCountDone, in2 := 2)
      I_Contact( "MvSkid_1".xREQ )
      wire#w1
      Move(in := 0, out1 => "MvSkid_1".MBmode)
   END_RUNG
   RUNG wire#w1
      Move(in := 40000, out1 => "MvSkid_1".MBdataAddr)
   END_RUNG
   RUNG wire#w1
      Move(in := 5, out1 => "MvSkid_1".MBdataLen)
   END_RUNG
   // the same network as SCL:
   IF ("MvSkid_1".iCountDone = 2) AND NOT "MvSkid_1".xREQ THEN
       "MvSkid_1".MBmode := 0;
       "MvSkid_1".MBdataAddr := 40000;
       "MvSkid_1".MBdataLen := 5;
   END_IF;
END_REGION

REGION Network 10: Read R_MVSKID data value
   // Select data coming from modbus
   RUNG wire#powerrail
      { S7_Templates := "SrcType := Int" } EQ_Contact(in1 := "MvSkid_1".iCountRead, in2 := 2)
      I_Contact( "MvSkid_1".xREQ )
      "PE_R_MVSKID"(Input_Data := "MvSkid_1".arrData, Output_Data => "MvSkid_1".R)
   END_RUNG
   // the same network as SCL:
   IF ("MvSkid_1".iCountRead = 2) AND NOT "MvSkid_1".xREQ THEN
       "PE_R_MVSKID"(Input_Data := "MvSkid_1".arrData, Output_Data => "MvSkid_1".R);
   END_IF;
END_REGION

REGION Network 11: U13.DI0.5
   // chiedere cosa signfica questi titoli
   RUNG wire#powerrail
      Contact( "PN".MVSKID.xCircBrkCloseCmd )
      Coil( "MvSkid_1".W.xCircBrk1CloseCmd )
   END_RUNG
   // the same network as SCL:
   "MvSkid_1".W.xCircBrk1CloseCmd := "PN".MVSKID.xCircBrkCloseCmd;
END_REGION

REGION Network 12: U13.DI0.4
   RUNG wire#powerrail
      Contact( "PN".MVSKID.xCircBrkOpenCmd )
      wire#w1
      Coil( "MvSkid_1".W.xCircBrk1OpenCmd )
   END_RUNG
   RUNG wire#powerrail
      Contact( "SM1".xMVbreakerOpenCmd )
   END_RUNG wire#w1
   RUNG wire#powerrail
      Contact( "SM2".xMVbreakerOpenCmd )
   END_RUNG wire#w1
   // the same network as SCL:
   "MvSkid_1".W.xCircBrk1OpenCmd := "PN".MVSKID.xCircBrkOpenCmd OR "SM1".xMVbreakerOpenCmd OR "SM2".xMVbreakerOpenCmd;
END_REGION

REGION Network 13: MV SKID Fault
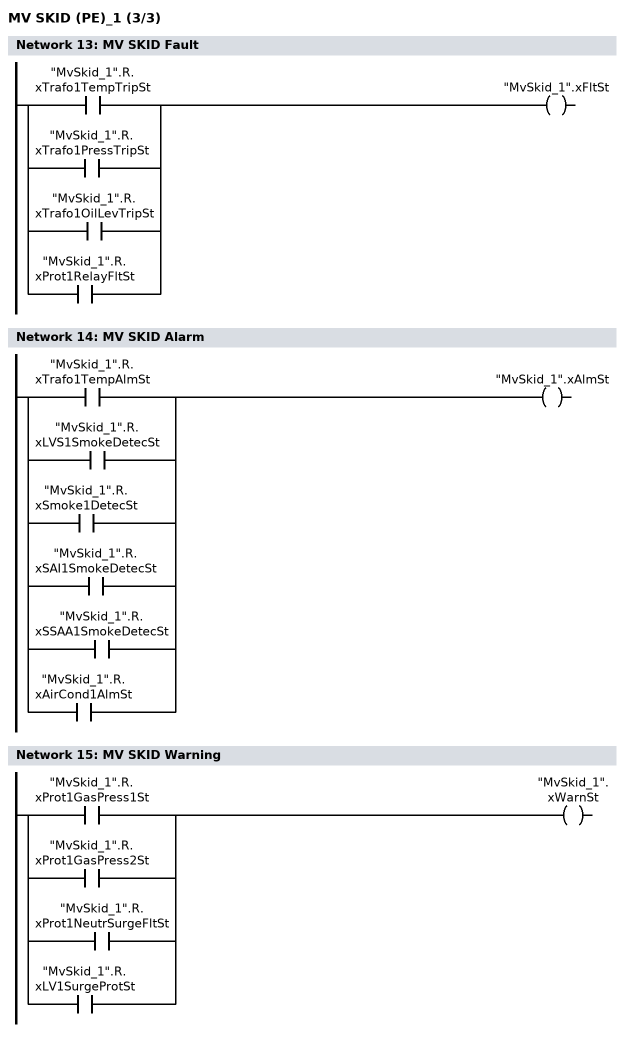
   RUNG wire#powerrail
      Contact( "MvSkid_1".R.xTrafo1TempTripSt )
      wire#w1
      Coil( "MvSkid_1".xFltSt )
   END_RUNG
   RUNG wire#powerrail
      Contact( "MvSkid_1".R.xTrafo1PressTripSt )
   END_RUNG wire#w1
   RUNG wire#powerrail
      Contact( "MvSkid_1".R.xTrafo1OilLevTripSt )
   END_RUNG wire#w1
   RUNG wire#powerrail
      Contact( "MvSkid_1".R.xProt1RelayFltSt )
   END_RUNG wire#w1
   // the same network as SCL:
   "MvSkid_1".xFltSt := "MvSkid_1".R.xTrafo1TempTripSt OR "MvSkid_1".R.xTrafo1PressTripSt OR "MvSkid_1".R.xTrafo1OilLevTripSt OR "MvSkid_1".R.xProt1RelayFltSt;
END_REGION

REGION Network 14: MV SKID Alarm
   RUNG wire#powerrail
      Contact( "MvSkid_1".R.xTrafo1TempAlmSt )
      wire#w1
      Coil( "MvSkid_1".xAlmSt )
   END_RUNG
   RUNG wire#powerrail
      Contact( "MvSkid_1".R.xLVS1SmokeDetecSt )
   END_RUNG wire#w1
   RUNG wire#powerrail
      Contact( "MvSkid_1".R.xSmoke1DetecSt )
   END_RUNG wire#w1
   RUNG wire#powerrail
      Contact( "MvSkid_1".R.xSAI1SmokeDetecSt )
   END_RUNG wire#w1
   RUNG wire#powerrail
      Contact( "MvSkid_1".R.xSSAA1SmokeDetecSt )
   END_RUNG wire#w1
   RUNG wire#powerrail
      Contact( "MvSkid_1".R.xAirCond1AlmSt )
   END_RUNG wire#w1
   // the same network as SCL:
   "MvSkid_1".xAlmSt := "MvSkid_1".R.xTrafo1TempAlmSt OR "MvSkid_1".R.xLVS1SmokeDetecSt OR "MvSkid_1".R.xSmoke1DetecSt OR "MvSkid_1".R.xSAI1SmokeDetecSt OR "MvSkid_1".R.xSSAA1SmokeDetecSt OR "MvSkid_1".R.xAirCond1AlmSt;
END_REGION

REGION Network 15: MV SKID Warning
   RUNG wire#powerrail
      Contact( "MvSkid_1".R.xProt1GasPress1St )
      wire#w1
      Coil( "MvSkid_1".xWarnSt )
   END_RUNG
   RUNG wire#powerrail
      Contact( "MvSkid_1".R.xProt1GasPress2St )
   END_RUNG wire#w1
   RUNG wire#powerrail
      Contact( "MvSkid_1".R.xProt1NeutrSurgeFltSt )
   END_RUNG wire#w1
   RUNG wire#powerrail
      Contact( "MvSkid_1".R.xLV1SurgeProtSt )
   END_RUNG wire#w1
   // the same network as SCL:
   "MvSkid_1".xWarnSt := "MvSkid_1".R.xProt1GasPress1St OR "MvSkid_1".R.xProt1GasPress2St OR "MvSkid_1".R.xProt1NeutrSurgeFltSt OR "MvSkid_1".R.xLV1SurgeProtSt;
END_REGION

REGION Network 16 (SCL): MV SKID Line Disconnector & Breaker Status
   "MvSkid_1".wLine1DiscSt.%X0 := "MvSkid_1".R.xLine1DiscOpenSt;
   "MvSkid_1".wLine1DiscSt.%X1 := "MvSkid_1".R.xLine1DiscCloseSt;
   "MvSkid_1".wLine1DiscSt.%X2 := "MvSkid_1".R.xLine1GndCloseSt;

   "MvSkid_1".wLine2DiscSt.%X0 := "MvSkid_1".R.xLine2DiscOpenSt;
   "MvSkid_1".wLine2DiscSt.%X1 := "MvSkid_1".R.xLine2DiscCloseSt;
   "MvSkid_1".wLine2DiscSt.%X2 := "MvSkid_1".R.xLine2GndCloseSt;

   "MvSkid_1".wProt1DiscSt.%X0 := "MvSkid_1".R.xProt1DiscOpenSt;
   "MvSkid_1".wProt1DiscSt.%X1 := "MvSkid_1".R.xProt1DiscCloseSt;
   "MvSkid_1".wProt1DiscSt.%X2 := "MvSkid_1".R.xProt1GndCloseSt;

   "MvSkid_1".wProt1CircBrkSt.%X0 := "MvSkid_1".R.xProt1CircBrkOpenSt;
   "MvSkid_1".wProt1CircBrkSt.%X1 := "MvSkid_1".R.xProt1CircBrkCloseSt;
END_REGION
END_FUNCTION

FUNCTION "PCS Faults_1" : Void   // FC43, LAD
{ S7_Optimized_Access := 'TRUE' }
VERSION : 0.1
// stored: AutoNumber false, IsIECCheckEnabled false, SetENOAutomatically false, UDAEnableTagReadback false
   VAR_TEMP
      wMF1 : Word;
      wMF2 : Word;
      wMF3 : Word;
      wMF4 : Word;
      wMW1 : Word;
      wMW2 : Word;
      wMW3 : Word;
      wMW4 : Word;
   END_VAR
   VAR_TEMP   // added for the SCL form of the ladder/FBD networks
      _w1 : Bool;
      _w2 : Bool;
      _w3 : Bool;
      _w4 : Bool;
   END_VAR
BEGIN

REGION Network 1: Split Inverter fault & warning and Module number - da eliminare
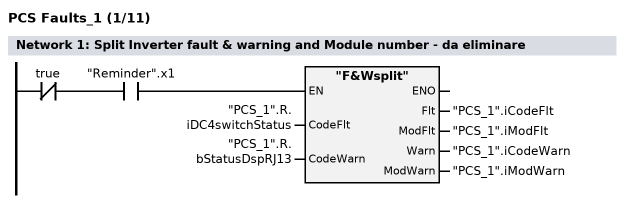
   RUNG wire#powerrail
      I_Contact( true )
      Contact( "Reminder".x1 )
      "F&Wsplit"(CodeFlt := "PCS_1".R.iDC4switchStatus, CodeWarn := "PCS_1".R.bStatusDspRJ13, Flt => "PCS_1".iCodeFlt, ModFlt => "PCS_1".iModFlt, Warn => "PCS_1".iCodeWarn, ModWarn => "PCS_1".iModWarn)
   END_RUNG
   // the same network as SCL:
   IF NOT true AND "Reminder".x1 THEN
       "F&Wsplit"(CodeFlt := "PCS_1".R.iDC4switchStatus,
                  CodeWarn := "PCS_1".R.bStatusDspRJ13,
                  Flt => "PCS_1".iCodeFlt,
                  ModFlt => "PCS_1".iModFlt,
                  Warn => "PCS_1".iCodeWarn,
                  ModWarn => "PCS_1".iModWarn);
   END_IF;
END_REGION

REGION Network 2: Inverter Faults
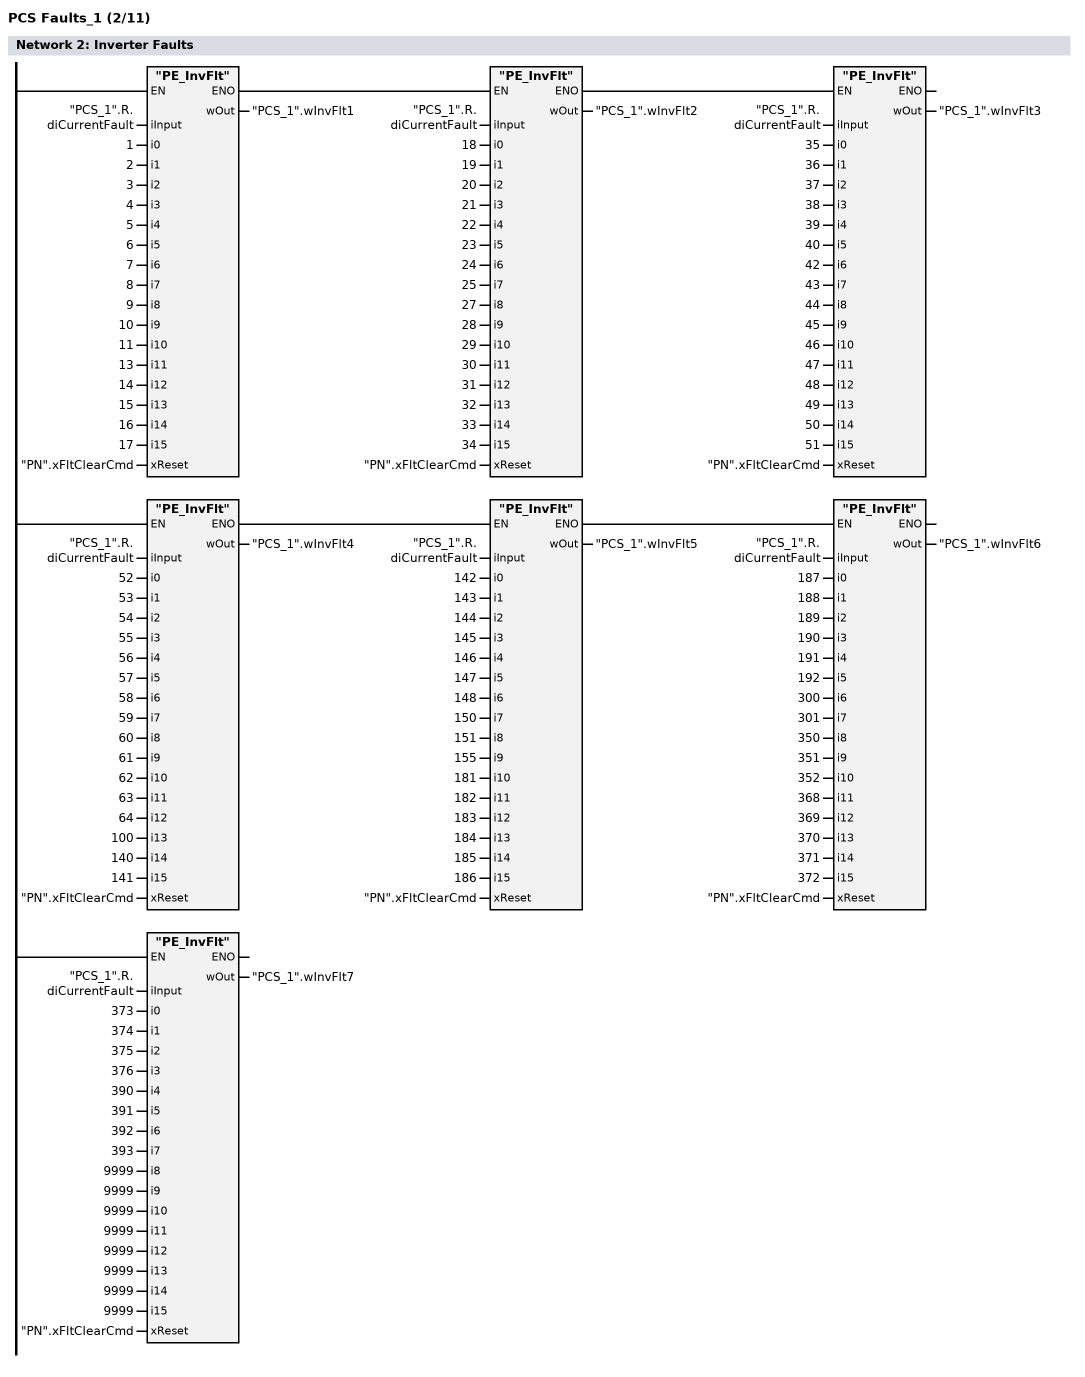
   RUNG wire#powerrail
      "PE_InvFlt"(iInput := "PCS_1".R.diCurrentFault, i0 := 1, i1 := 2, i2 := 3, i3 := 4, i4 := 5, i5 := 6, i6 := 7, i7 := 8, i8 := 9, i9 := 10, i10 := 11, i11 := 13, i12 := 14, i13 := 15, i14 := 16, i15 := 17, xReset := "PN".xFltClearCmd, wOut => "PCS_1".wInvFlt1)
      "PE_InvFlt"(iInput := "PCS_1".R.diCurrentFault, i0 := 18, i1 := 19, i2 := 20, i3 := 21, i4 := 22, i5 := 23, i6 := 24, i7 := 25, i8 := 27, i9 := 28, i10 := 29, i11 := 30, i12 := 31, i13 := 32, i14 := 33, i15 := 34, xReset := "PN".xFltClearCmd, wOut => "PCS_1".wInvFlt2)
      "PE_InvFlt"(iInput := "PCS_1".R.diCurrentFault, i0 := 35, i1 := 36, i2 := 37, i3 := 38, i4 := 39, i5 := 40, i6 := 42, i7 := 43, i8 := 44, i9 := 45, i10 := 46, i11 := 47, i12 := 48, i13 := 49, i14 := 50, i15 := 51, xReset := "PN".xFltClearCmd, wOut => "PCS_1".wInvFlt3)
   END_RUNG
   RUNG wire#powerrail
      "PE_InvFlt"(iInput := "PCS_1".R.diCurrentFault, i0 := 52, i1 := 53, i2 := 54, i3 := 55, i4 := 56, i5 := 57, i6 := 58, i7 := 59, i8 := 60, i9 := 61, i10 := 62, i11 := 63, i12 := 64, i13 := 100, i14 := 140, i15 := 141, xReset := "PN".xFltClearCmd, wOut => "PCS_1".wInvFlt4)
      "PE_InvFlt"(iInput := "PCS_1".R.diCurrentFault, i0 := 142, i1 := 143, i2 := 144, i3 := 145, i4 := 146, i5 := 147, i6 := 148, i7 := 150, i8 := 151, i9 := 155, i10 := 181, i11 := 182, i12 := 183, i13 := 184, i14 := 185, i15 := 186, xReset := "PN".xFltClearCmd, wOut => "PCS_1".wInvFlt5)
      "PE_InvFlt"(iInput := "PCS_1".R.diCurrentFault, i0 := 187, i1 := 188, i2 := 189, i3 := 190, i4 := 191, i5 := 192, i6 := 300, i7 := 301, i8 := 350, i9 := 351, i10 := 352, i11 := 368, i12 := 369, i13 := 370, i14 := 371, i15 := 372, xReset := "PN".xFltClearCmd, wOut => "PCS_1".wInvFlt6)
   END_RUNG
   RUNG wire#powerrail
      "PE_InvFlt"(iInput := "PCS_1".R.diCurrentFault, i0 := 373, i1 := 374, i2 := 375, i3 := 376, i4 := 390, i5 := 391, i6 := 392, i7 := 393, i8 := 9999, i9 := 9999, i10 := 9999, i11 := 9999, i12 := 9999, i13 := 9999, i14 := 9999, i15 := 9999, xReset := "PN".xFltClearCmd, wOut => "PCS_1".wInvFlt7)
   END_RUNG
   // the same network as SCL:
   "PE_InvFlt"(iInput := "PCS_1".R.diCurrentFault,
               i0 := 1,
               i1 := 2,
               i2 := 3,
               i3 := 4,
               i4 := 5,
               i5 := 6,
               i6 := 7,
               i7 := 8,
               i8 := 9,
               i9 := 10,
               i10 := 11,
               i11 := 13,
               i12 := 14,
               i13 := 15,
               i14 := 16,
               i15 := 17,
               xReset := "PN".xFltClearCmd,
               wOut => "PCS_1".wInvFlt1,
               ENO => #_w1);
   "PE_InvFlt"(EN := #_w1,
               iInput := "PCS_1".R.diCurrentFault,
               i0 := 18,
               i1 := 19,
               i2 := 20,
               i3 := 21,
               i4 := 22,
               i5 := 23,
               i6 := 24,
               i7 := 25,
               i8 := 27,
               i9 := 28,
               i10 := 29,
               i11 := 30,
               i12 := 31,
               i13 := 32,
               i14 := 33,
               i15 := 34,
               xReset := "PN".xFltClearCmd,
               wOut => "PCS_1".wInvFlt2,
               ENO => #_w2);
   IF #_w2 THEN
       "PE_InvFlt"(iInput := "PCS_1".R.diCurrentFault,
                   i0 := 35,
                   i1 := 36,
                   i2 := 37,
                   i3 := 38,
                   i4 := 39,
                   i5 := 40,
                   i6 := 42,
                   i7 := 43,
                   i8 := 44,
                   i9 := 45,
                   i10 := 46,
                   i11 := 47,
                   i12 := 48,
                   i13 := 49,
                   i14 := 50,
                   i15 := 51,
                   xReset := "PN".xFltClearCmd,
                   wOut => "PCS_1".wInvFlt3);
   END_IF;
   "PE_InvFlt"(iInput := "PCS_1".R.diCurrentFault,
               i0 := 52,
               i1 := 53,
               i2 := 54,
               i3 := 55,
               i4 := 56,
               i5 := 57,
               i6 := 58,
               i7 := 59,
               i8 := 60,
               i9 := 61,
               i10 := 62,
               i11 := 63,
               i12 := 64,
               i13 := 100,
               i14 := 140,
               i15 := 141,
               xReset := "PN".xFltClearCmd,
               wOut => "PCS_1".wInvFlt4,
               ENO => #_w3);
   "PE_InvFlt"(EN := #_w3,
               iInput := "PCS_1".R.diCurrentFault,
               i0 := 142,
               i1 := 143,
               i2 := 144,
               i3 := 145,
               i4 := 146,
               i5 := 147,
               i6 := 148,
               i7 := 150,
               i8 := 151,
               i9 := 155,
               i10 := 181,
               i11 := 182,
               i12 := 183,
               i13 := 184,
               i14 := 185,
               i15 := 186,
               xReset := "PN".xFltClearCmd,
               wOut => "PCS_1".wInvFlt5,
               ENO => #_w4);
   IF #_w4 THEN
       "PE_InvFlt"(iInput := "PCS_1".R.diCurrentFault,
                   i0 := 187,
                   i1 := 188,
                   i2 := 189,
                   i3 := 190,
                   i4 := 191,
                   i5 := 192,
                   i6 := 300,
                   i7 := 301,
                   i8 := 350,
                   i9 := 351,
                   i10 := 352,
                   i11 := 368,
                   i12 := 369,
                   i13 := 370,
                   i14 := 371,
                   i15 := 372,
                   xReset := "PN".xFltClearCmd,
                   wOut => "PCS_1".wInvFlt6);
   END_IF;
   "PE_InvFlt"(iInput := "PCS_1".R.diCurrentFault,
               i0 := 373,
               i1 := 374,
               i2 := 375,
               i3 := 376,
               i4 := 390,
               i5 := 391,
               i6 := 392,
               i7 := 393,
               i8 := 9999,
               i9 := 9999,
               i10 := 9999,
               i11 := 9999,
               i12 := 9999,
               i13 := 9999,
               i14 := 9999,
               i15 := 9999,
               xReset := "PN".xFltClearCmd,
               wOut => "PCS_1".wInvFlt7);
END_REGION

REGION Network 3: Inverter Warning
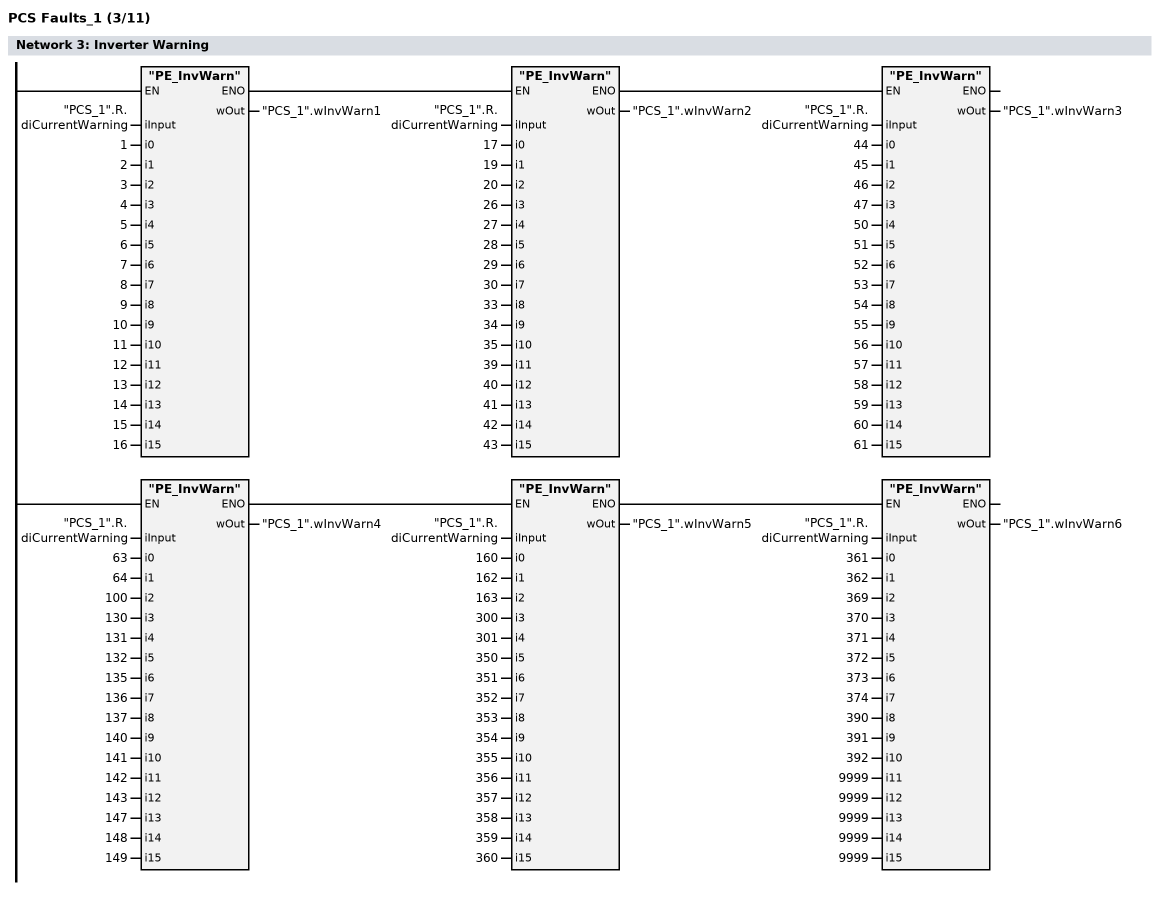
   RUNG wire#powerrail
      "PE_InvWarn"(iInput := "PCS_1".R.diCurrentWarning, i0 := 1, i1 := 2, i2 := 3, i3 := 4, i4 := 5, i5 := 6, i6 := 7, i7 := 8, i8 := 9, i9 := 10, i10 := 11, i11 := 12, i12 := 13, i13 := 14, i14 := 15, i15 := 16, wOut => "PCS_1".wInvWarn1)
      "PE_InvWarn"(iInput := "PCS_1".R.diCurrentWarning, i0 := 17, i1 := 19, i2 := 20, i3 := 26, i4 := 27, i5 := 28, i6 := 29, i7 := 30, i8 := 33, i9 := 34, i10 := 35, i11 := 39, i12 := 40, i13 := 41, i14 := 42, i15 := 43, wOut => "PCS_1".wInvWarn2)
      "PE_InvWarn"(iInput := "PCS_1".R.diCurrentWarning, i0 := 44, i1 := 45, i2 := 46, i3 := 47, i4 := 50, i5 := 51, i6 := 52, i7 := 53, i8 := 54, i9 := 55, i10 := 56, i11 := 57, i12 := 58, i13 := 59, i14 := 60, i15 := 61, wOut => "PCS_1".wInvWarn3)
   END_RUNG
   RUNG wire#powerrail
      "PE_InvWarn"(iInput := "PCS_1".R.diCurrentWarning, i0 := 63, i1 := 64, i2 := 100, i3 := 130, i4 := 131, i5 := 132, i6 := 135, i7 := 136, i8 := 137, i9 := 140, i10 := 141, i11 := 142, i12 := 143, i13 := 147, i14 := 148, i15 := 149, wOut => "PCS_1".wInvWarn4)
      "PE_InvWarn"(iInput := "PCS_1".R.diCurrentWarning, i0 := 160, i1 := 162, i2 := 163, i3 := 300, i4 := 301, i5 := 350, i6 := 351, i7 := 352, i8 := 353, i9 := 354, i10 := 355, i11 := 356, i12 := 357, i13 := 358, i14 := 359, i15 := 360, wOut => "PCS_1".wInvWarn5)
      "PE_InvWarn"(iInput := "PCS_1".R.diCurrentWarning, i0 := 361, i1 := 362, i2 := 369, i3 := 370, i4 := 371, i5 := 372, i6 := 373, i7 := 374, i8 := 390, i9 := 391, i10 := 392, i11 := 9999, i12 := 9999, i13 := 9999, i14 := 9999, i15 := 9999, wOut => "PCS_1".wInvWarn6)
   END_RUNG
   // the same network as SCL:
   "PE_InvWarn"(iInput := "PCS_1".R.diCurrentWarning,
                i0 := 1,
                i1 := 2,
                i2 := 3,
                i3 := 4,
                i4 := 5,
                i5 := 6,
                i6 := 7,
                i7 := 8,
                i8 := 9,
                i9 := 10,
                i10 := 11,
                i11 := 12,
                i12 := 13,
                i13 := 14,
                i14 := 15,
                i15 := 16,
                wOut => "PCS_1".wInvWarn1,
                ENO => #_w1);
   "PE_InvWarn"(EN := #_w1,
                iInput := "PCS_1".R.diCurrentWarning,
                i0 := 17,
                i1 := 19,
                i2 := 20,
                i3 := 26,
                i4 := 27,
                i5 := 28,
                i6 := 29,
                i7 := 30,
                i8 := 33,
                i9 := 34,
                i10 := 35,
                i11 := 39,
                i12 := 40,
                i13 := 41,
                i14 := 42,
                i15 := 43,
                wOut => "PCS_1".wInvWarn2,
                ENO => #_w2);
   IF #_w2 THEN
       "PE_InvWarn"(iInput := "PCS_1".R.diCurrentWarning,
                    i0 := 44,
                    i1 := 45,
                    i2 := 46,
                    i3 := 47,
                    i4 := 50,
                    i5 := 51,
                    i6 := 52,
                    i7 := 53,
                    i8 := 54,
                    i9 := 55,
                    i10 := 56,
                    i11 := 57,
                    i12 := 58,
                    i13 := 59,
                    i14 := 60,
                    i15 := 61,
                    wOut => "PCS_1".wInvWarn3);
   END_IF;
   "PE_InvWarn"(iInput := "PCS_1".R.diCurrentWarning,
                i0 := 63,
                i1 := 64,
                i2 := 100,
                i3 := 130,
                i4 := 131,
                i5 := 132,
                i6 := 135,
                i7 := 136,
                i8 := 137,
                i9 := 140,
                i10 := 141,
                i11 := 142,
                i12 := 143,
                i13 := 147,
                i14 := 148,
                i15 := 149,
                wOut => "PCS_1".wInvWarn4,
                ENO => #_w3);
   "PE_InvWarn"(EN := #_w3,
                iInput := "PCS_1".R.diCurrentWarning,
                i0 := 160,
                i1 := 162,
                i2 := 163,
                i3 := 300,
                i4 := 301,
                i5 := 350,
                i6 := 351,
                i7 := 352,
                i8 := 353,
                i9 := 354,
                i10 := 355,
                i11 := 356,
                i12 := 357,
                i13 := 358,
                i14 := 359,
                i15 := 360,
                wOut => "PCS_1".wInvWarn5,
                ENO => #_w4);
   IF #_w4 THEN
       "PE_InvWarn"(iInput := "PCS_1".R.diCurrentWarning,
                    i0 := 361,
                    i1 := 362,
                    i2 := 369,
                    i3 := 370,
                    i4 := 371,
                    i5 := 372,
                    i6 := 373,
                    i7 := 374,
                    i8 := 390,
                    i9 := 391,
                    i10 := 392,
                    i11 := 9999,
                    i12 := 9999,
                    i13 := 9999,
                    i14 := 9999,
                    i15 := 9999,
                    wOut => "PCS_1".wInvWarn6);
   END_IF;
END_REGION

REGION Network 4: Module Faults
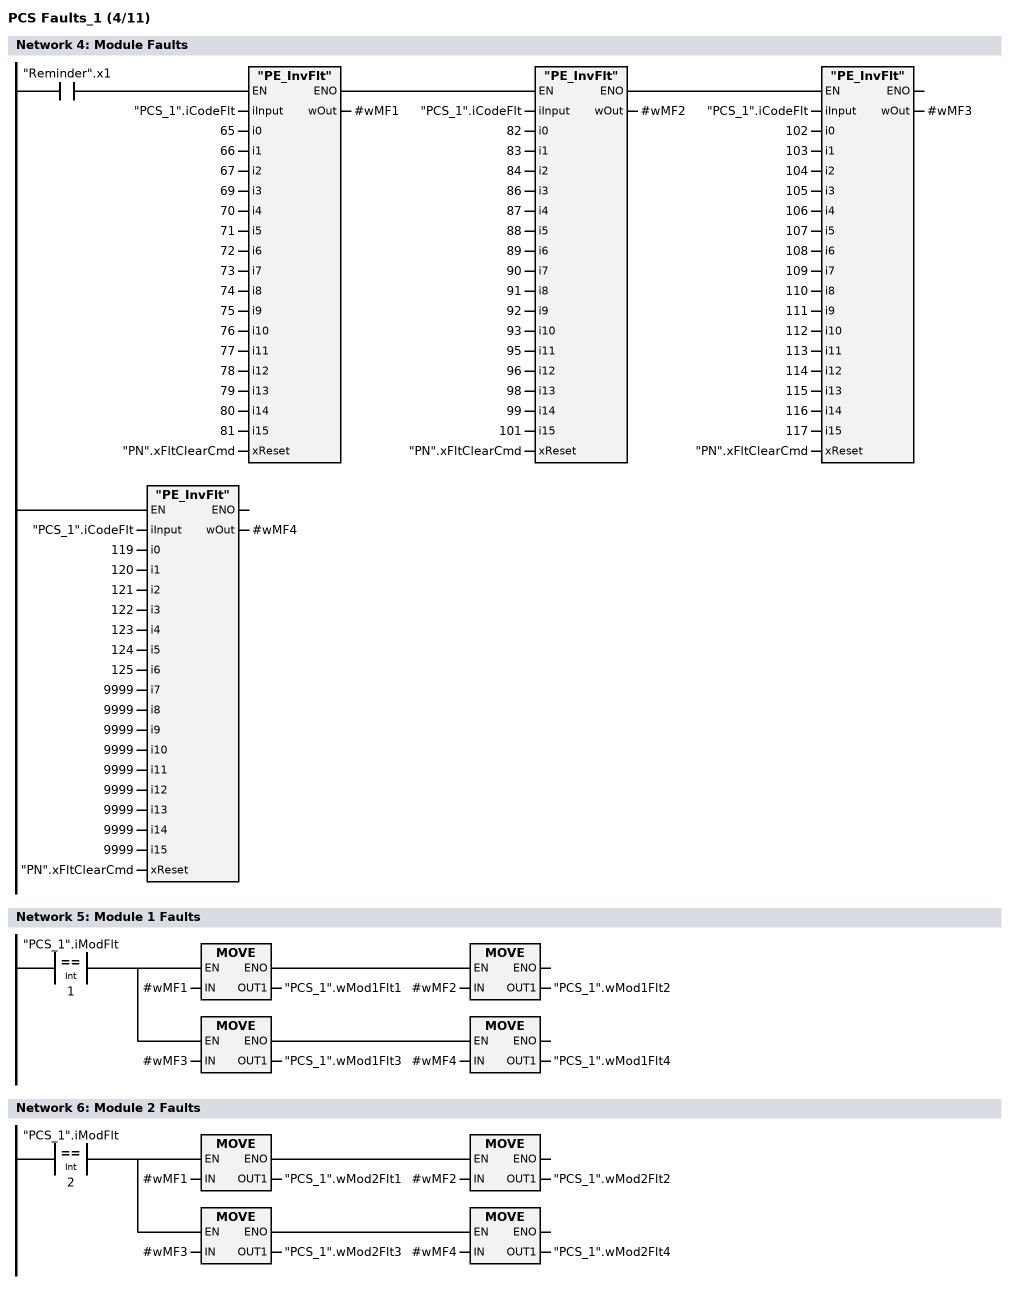
   RUNG wire#powerrail
      Contact( "Reminder".x1 )
      "PE_InvFlt"(iInput := "PCS_1".iCodeFlt, i0 := 65, i1 := 66, i2 := 67, i3 := 69, i4 := 70, i5 := 71, i6 := 72, i7 := 73, i8 := 74, i9 := 75, i10 := 76, i11 := 77, i12 := 78, i13 := 79, i14 := 80, i15 := 81, xReset := "PN".xFltClearCmd, wOut => #wMF1)
      "PE_InvFlt"(iInput := "PCS_1".iCodeFlt, i0 := 82, i1 := 83, i2 := 84, i3 := 86, i4 := 87, i5 := 88, i6 := 89, i7 := 90, i8 := 91, i9 := 92, i10 := 93, i11 := 95, i12 := 96, i13 := 98, i14 := 99, i15 := 101, xReset := "PN".xFltClearCmd, wOut => #wMF2)
      "PE_InvFlt"(iInput := "PCS_1".iCodeFlt, i0 := 102, i1 := 103, i2 := 104, i3 := 105, i4 := 106, i5 := 107, i6 := 108, i7 := 109, i8 := 110, i9 := 111, i10 := 112, i11 := 113, i12 := 114, i13 := 115, i14 := 116, i15 := 117, xReset := "PN".xFltClearCmd, wOut => #wMF3)
   END_RUNG
   RUNG wire#powerrail
      "PE_InvFlt"(iInput := "PCS_1".iCodeFlt, i0 := 119, i1 := 120, i2 := 121, i3 := 122, i4 := 123, i5 := 124, i6 := 125, i7 := 9999, i8 := 9999, i9 := 9999, i10 := 9999, i11 := 9999, i12 := 9999, i13 := 9999, i14 := 9999, i15 := 9999, xReset := "PN".xFltClearCmd, wOut => #wMF4)
   END_RUNG
   // the same network as SCL:
   "PE_InvFlt"(EN := "Reminder".x1,
               iInput := "PCS_1".iCodeFlt,
               i0 := 65,
               i1 := 66,
               i2 := 67,
               i3 := 69,
               i4 := 70,
               i5 := 71,
               i6 := 72,
               i7 := 73,
               i8 := 74,
               i9 := 75,
               i10 := 76,
               i11 := 77,
               i12 := 78,
               i13 := 79,
               i14 := 80,
               i15 := 81,
               xReset := "PN".xFltClearCmd,
               wOut => #wMF1,
               ENO => #_w1);
   "PE_InvFlt"(EN := #_w1,
               iInput := "PCS_1".iCodeFlt,
               i0 := 82,
               i1 := 83,
               i2 := 84,
               i3 := 86,
               i4 := 87,
               i5 := 88,
               i6 := 89,
               i7 := 90,
               i8 := 91,
               i9 := 92,
               i10 := 93,
               i11 := 95,
               i12 := 96,
               i13 := 98,
               i14 := 99,
               i15 := 101,
               xReset := "PN".xFltClearCmd,
               wOut => #wMF2,
               ENO => #_w2);
   IF #_w2 THEN
       "PE_InvFlt"(iInput := "PCS_1".iCodeFlt,
                   i0 := 102,
                   i1 := 103,
                   i2 := 104,
                   i3 := 105,
                   i4 := 106,
                   i5 := 107,
                   i6 := 108,
                   i7 := 109,
                   i8 := 110,
                   i9 := 111,
                   i10 := 112,
                   i11 := 113,
                   i12 := 114,
                   i13 := 115,
                   i14 := 116,
                   i15 := 117,
                   xReset := "PN".xFltClearCmd,
                   wOut => #wMF3);
   END_IF;
   "PE_InvFlt"(iInput := "PCS_1".iCodeFlt,
               i0 := 119,
               i1 := 120,
               i2 := 121,
               i3 := 122,
               i4 := 123,
               i5 := 124,
               i6 := 125,
               i7 := 9999,
               i8 := 9999,
               i9 := 9999,
               i10 := 9999,
               i11 := 9999,
               i12 := 9999,
               i13 := 9999,
               i14 := 9999,
               i15 := 9999,
               xReset := "PN".xFltClearCmd,
               wOut => #wMF4);
END_REGION

REGION Network 5: Module 1 Faults
   RUNG wire#powerrail
      { S7_Templates := "SrcType := Int" } EQ_Contact(in1 := "PCS_1".iModFlt, in2 := 1)
      wire#w1
      Move(in := #wMF1, out1 => "PCS_1".wMod1Flt1)
      Move(in := #wMF2, out1 => "PCS_1".wMod1Flt2)
   END_RUNG
   RUNG wire#w1
      Move(in := #wMF3, out1 => "PCS_1".wMod1Flt3)
      Move(in := #wMF4, out1 => "PCS_1".wMod1Flt4)
   END_RUNG
   // the same network as SCL:
   IF "PCS_1".iModFlt = 1 THEN
       "PCS_1".wMod1Flt1 := #wMF1;
       "PCS_1".wMod1Flt2 := #wMF2;
       "PCS_1".wMod1Flt3 := #wMF3;
       "PCS_1".wMod1Flt4 := #wMF4;
   END_IF;
END_REGION

REGION Network 6: Module 2 Faults
   RUNG wire#powerrail
      { S7_Templates := "SrcType := Int" } EQ_Contact(in1 := "PCS_1".iModFlt, in2 := 2)
      wire#w1
      Move(in := #wMF1, out1 => "PCS_1".wMod2Flt1)
      Move(in := #wMF2, out1 => "PCS_1".wMod2Flt2)
   END_RUNG
   RUNG wire#w1
      Move(in := #wMF3, out1 => "PCS_1".wMod2Flt3)
      Move(in := #wMF4, out1 => "PCS_1".wMod2Flt4)
   END_RUNG
   // the same network as SCL:
   IF "PCS_1".iModFlt = 2 THEN
       "PCS_1".wMod2Flt1 := #wMF1;
       "PCS_1".wMod2Flt2 := #wMF2;
       "PCS_1".wMod2Flt3 := #wMF3;
       "PCS_1".wMod2Flt4 := #wMF4;
   END_IF;
END_REGION

REGION Network 7: Module 3 Faults
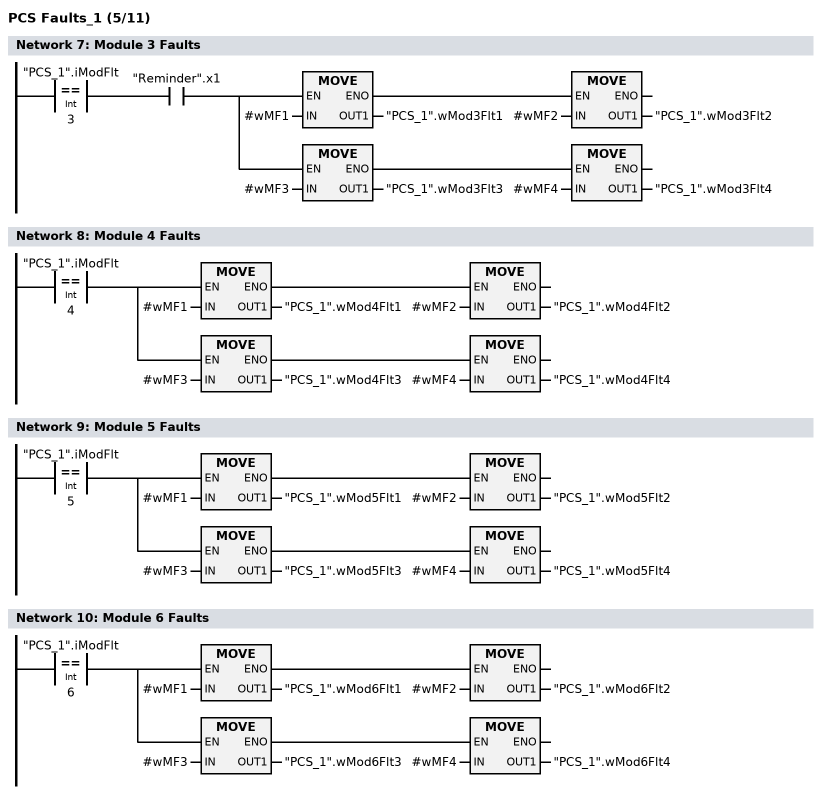
   RUNG wire#powerrail
      { S7_Templates := "SrcType := Int" } EQ_Contact(in1 := "PCS_1".iModFlt, in2 := 3)
      Contact( "Reminder".x1 )
      wire#w1
      Move(in := #wMF1, out1 => "PCS_1".wMod3Flt1)
      Move(in := #wMF2, out1 => "PCS_1".wMod3Flt2)
   END_RUNG
   RUNG wire#w1
      Move(in := #wMF3, out1 => "PCS_1".wMod3Flt3)
      Move(in := #wMF4, out1 => "PCS_1".wMod3Flt4)
   END_RUNG
   // the same network as SCL:
   IF ("PCS_1".iModFlt = 3) AND "Reminder".x1 THEN
       "PCS_1".wMod3Flt1 := #wMF1;
       "PCS_1".wMod3Flt2 := #wMF2;
       "PCS_1".wMod3Flt3 := #wMF3;
       "PCS_1".wMod3Flt4 := #wMF4;
   END_IF;
END_REGION

REGION Network 8: Module 4 Faults
   RUNG wire#powerrail
      { S7_Templates := "SrcType := Int" } EQ_Contact(in1 := "PCS_1".iModFlt, in2 := 4)
      wire#w1
      Move(in := #wMF1, out1 => "PCS_1".wMod4Flt1)
      Move(in := #wMF2, out1 => "PCS_1".wMod4Flt2)
   END_RUNG
   RUNG wire#w1
      Move(in := #wMF3, out1 => "PCS_1".wMod4Flt3)
      Move(in := #wMF4, out1 => "PCS_1".wMod4Flt4)
   END_RUNG
   // the same network as SCL:
   IF "PCS_1".iModFlt = 4 THEN
       "PCS_1".wMod4Flt1 := #wMF1;
       "PCS_1".wMod4Flt2 := #wMF2;
       "PCS_1".wMod4Flt3 := #wMF3;
       "PCS_1".wMod4Flt4 := #wMF4;
   END_IF;
END_REGION

REGION Network 9: Module 5 Faults
   RUNG wire#powerrail
      { S7_Templates := "SrcType := Int" } EQ_Contact(in1 := "PCS_1".iModFlt, in2 := 5)
      wire#w1
      Move(in := #wMF1, out1 => "PCS_1".wMod5Flt1)
      Move(in := #wMF2, out1 => "PCS_1".wMod5Flt2)
   END_RUNG
   RUNG wire#w1
      Move(in := #wMF3, out1 => "PCS_1".wMod5Flt3)
      Move(in := #wMF4, out1 => "PCS_1".wMod5Flt4)
   END_RUNG
   // the same network as SCL:
   IF "PCS_1".iModFlt = 5 THEN
       "PCS_1".wMod5Flt1 := #wMF1;
       "PCS_1".wMod5Flt2 := #wMF2;
       "PCS_1".wMod5Flt3 := #wMF3;
       "PCS_1".wMod5Flt4 := #wMF4;
   END_IF;
END_REGION

REGION Network 10: Module 6 Faults
   RUNG wire#powerrail
      { S7_Templates := "SrcType := Int" } EQ_Contact(in1 := "PCS_1".iModFlt, in2 := 6)
      wire#w1
      Move(in := #wMF1, out1 => "PCS_1".wMod6Flt1)
      Move(in := #wMF2, out1 => "PCS_1".wMod6Flt2)
   END_RUNG
   RUNG wire#w1
      Move(in := #wMF3, out1 => "PCS_1".wMod6Flt3)
      Move(in := #wMF4, out1 => "PCS_1".wMod6Flt4)
   END_RUNG
   // the same network as SCL:
   IF "PCS_1".iModFlt = 6 THEN
       "PCS_1".wMod6Flt1 := #wMF1;
       "PCS_1".wMod6Flt2 := #wMF2;
       "PCS_1".wMod6Flt3 := #wMF3;
       "PCS_1".wMod6Flt4 := #wMF4;
   END_IF;
END_REGION

REGION Network 11: Module Warnings
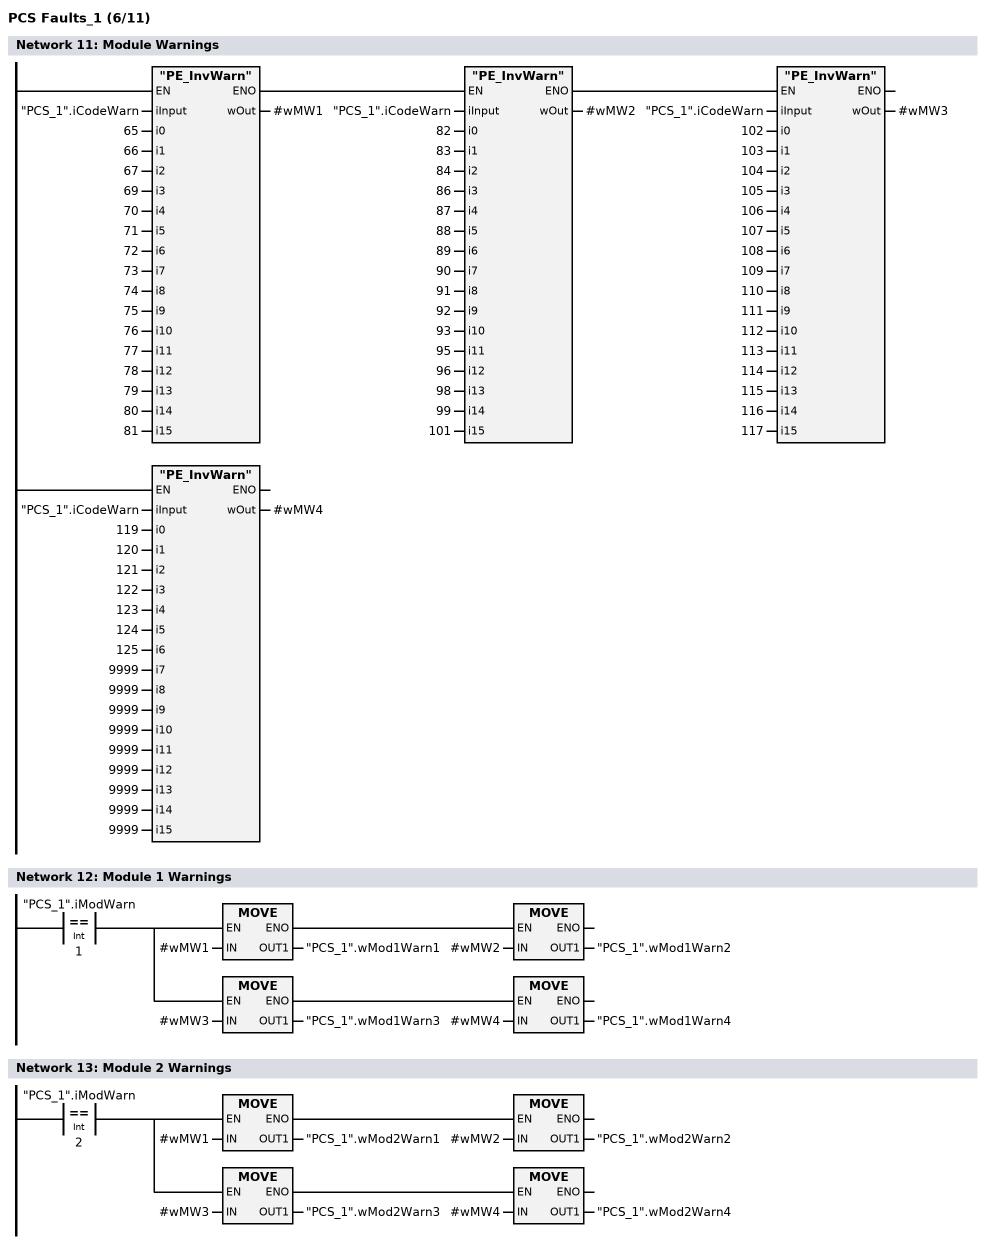
   RUNG wire#powerrail
      "PE_InvWarn"(iInput := "PCS_1".iCodeWarn, i0 := 65, i1 := 66, i2 := 67, i3 := 69, i4 := 70, i5 := 71, i6 := 72, i7 := 73, i8 := 74, i9 := 75, i10 := 76, i11 := 77, i12 := 78, i13 := 79, i14 := 80, i15 := 81, wOut => #wMW1)
      "PE_InvWarn"(iInput := "PCS_1".iCodeWarn, i0 := 82, i1 := 83, i2 := 84, i3 := 86, i4 := 87, i5 := 88, i6 := 89, i7 := 90, i8 := 91, i9 := 92, i10 := 93, i11 := 95, i12 := 96, i13 := 98, i14 := 99, i15 := 101, wOut => #wMW2)
      "PE_InvWarn"(iInput := "PCS_1".iCodeWarn, i0 := 102, i1 := 103, i2 := 104, i3 := 105, i4 := 106, i5 := 107, i6 := 108, i7 := 109, i8 := 110, i9 := 111, i10 := 112, i11 := 113, i12 := 114, i13 := 115, i14 := 116, i15 := 117, wOut => #wMW3)
   END_RUNG
   RUNG wire#powerrail
      "PE_InvWarn"(iInput := "PCS_1".iCodeWarn, i0 := 119, i1 := 120, i2 := 121, i3 := 122, i4 := 123, i5 := 124, i6 := 125, i7 := 9999, i8 := 9999, i9 := 9999, i10 := 9999, i11 := 9999, i12 := 9999, i13 := 9999, i14 := 9999, i15 := 9999, wOut => #wMW4)
   END_RUNG
   // the same network as SCL:
   "PE_InvWarn"(iInput := "PCS_1".iCodeWarn,
                i0 := 65,
                i1 := 66,
                i2 := 67,
                i3 := 69,
                i4 := 70,
                i5 := 71,
                i6 := 72,
                i7 := 73,
                i8 := 74,
                i9 := 75,
                i10 := 76,
                i11 := 77,
                i12 := 78,
                i13 := 79,
                i14 := 80,
                i15 := 81,
                wOut => #wMW1,
                ENO => #_w1);
   "PE_InvWarn"(EN := #_w1,
                iInput := "PCS_1".iCodeWarn,
                i0 := 82,
                i1 := 83,
                i2 := 84,
                i3 := 86,
                i4 := 87,
                i5 := 88,
                i6 := 89,
                i7 := 90,
                i8 := 91,
                i9 := 92,
                i10 := 93,
                i11 := 95,
                i12 := 96,
                i13 := 98,
                i14 := 99,
                i15 := 101,
                wOut => #wMW2,
                ENO => #_w2);
   IF #_w2 THEN
       "PE_InvWarn"(iInput := "PCS_1".iCodeWarn,
                    i0 := 102,
                    i1 := 103,
                    i2 := 104,
                    i3 := 105,
                    i4 := 106,
                    i5 := 107,
                    i6 := 108,
                    i7 := 109,
                    i8 := 110,
                    i9 := 111,
                    i10 := 112,
                    i11 := 113,
                    i12 := 114,
                    i13 := 115,
                    i14 := 116,
                    i15 := 117,
                    wOut => #wMW3);
   END_IF;
   "PE_InvWarn"(iInput := "PCS_1".iCodeWarn,
                i0 := 119,
                i1 := 120,
                i2 := 121,
                i3 := 122,
                i4 := 123,
                i5 := 124,
                i6 := 125,
                i7 := 9999,
                i8 := 9999,
                i9 := 9999,
                i10 := 9999,
                i11 := 9999,
                i12 := 9999,
                i13 := 9999,
                i14 := 9999,
                i15 := 9999,
                wOut => #wMW4);
END_REGION

REGION Network 12: Module 1 Warnings
   RUNG wire#powerrail
      { S7_Templates := "SrcType := Int" } EQ_Contact(in1 := "PCS_1".iModWarn, in2 := 1)
      wire#w1
      Move(in := #wMW1, out1 => "PCS_1".wMod1Warn1)
      Move(in := #wMW2, out1 => "PCS_1".wMod1Warn2)
   END_RUNG
   RUNG wire#w1
      Move(in := #wMW3, out1 => "PCS_1".wMod1Warn3)
      Move(in := #wMW4, out1 => "PCS_1".wMod1Warn4)
   END_RUNG
   // the same network as SCL:
   IF "PCS_1".iModWarn = 1 THEN
       "PCS_1".wMod1Warn1 := #wMW1;
       "PCS_1".wMod1Warn2 := #wMW2;
       "PCS_1".wMod1Warn3 := #wMW3;
       "PCS_1".wMod1Warn4 := #wMW4;
   END_IF;
END_REGION

REGION Network 13: Module 2 Warnings
   RUNG wire#powerrail
      { S7_Templates := "SrcType := Int" } EQ_Contact(in1 := "PCS_1".iModWarn, in2 := 2)
      wire#w1
      Move(in := #wMW1, out1 => "PCS_1".wMod2Warn1)
      Move(in := #wMW2, out1 => "PCS_1".wMod2Warn2)
   END_RUNG
   RUNG wire#w1
      Move(in := #wMW3, out1 => "PCS_1".wMod2Warn3)
      Move(in := #wMW4, out1 => "PCS_1".wMod2Warn4)
   END_RUNG
   // the same network as SCL:
   IF "PCS_1".iModWarn = 2 THEN
       "PCS_1".wMod2Warn1 := #wMW1;
       "PCS_1".wMod2Warn2 := #wMW2;
       "PCS_1".wMod2Warn3 := #wMW3;
       "PCS_1".wMod2Warn4 := #wMW4;
   END_IF;
END_REGION

REGION Network 14: Module 3 Warnings
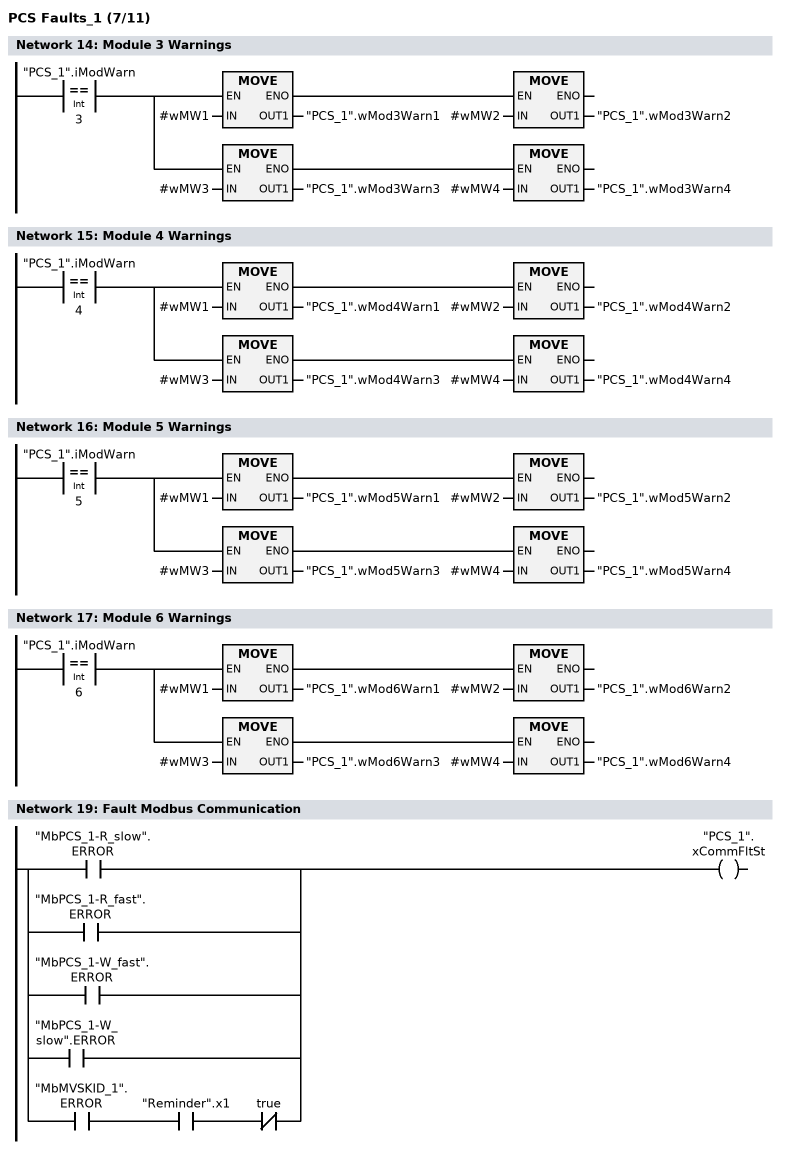
   RUNG wire#powerrail
      { S7_Templates := "SrcType := Int" } EQ_Contact(in1 := "PCS_1".iModWarn, in2 := 3)
      wire#w1
      Move(in := #wMW1, out1 => "PCS_1".wMod3Warn1)
      Move(in := #wMW2, out1 => "PCS_1".wMod3Warn2)
   END_RUNG
   RUNG wire#w1
      Move(in := #wMW3, out1 => "PCS_1".wMod3Warn3)
      Move(in := #wMW4, out1 => "PCS_1".wMod3Warn4)
   END_RUNG
   // the same network as SCL:
   IF "PCS_1".iModWarn = 3 THEN
       "PCS_1".wMod3Warn1 := #wMW1;
       "PCS_1".wMod3Warn2 := #wMW2;
       "PCS_1".wMod3Warn3 := #wMW3;
       "PCS_1".wMod3Warn4 := #wMW4;
   END_IF;
END_REGION

REGION Network 15: Module 4 Warnings
   RUNG wire#powerrail
      { S7_Templates := "SrcType := Int" } EQ_Contact(in1 := "PCS_1".iModWarn, in2 := 4)
      wire#w1
      Move(in := #wMW1, out1 => "PCS_1".wMod4Warn1)
      Move(in := #wMW2, out1 => "PCS_1".wMod4Warn2)
   END_RUNG
   RUNG wire#w1
      Move(in := #wMW3, out1 => "PCS_1".wMod4Warn3)
      Move(in := #wMW4, out1 => "PCS_1".wMod4Warn4)
   END_RUNG
   // the same network as SCL:
   IF "PCS_1".iModWarn = 4 THEN
       "PCS_1".wMod4Warn1 := #wMW1;
       "PCS_1".wMod4Warn2 := #wMW2;
       "PCS_1".wMod4Warn3 := #wMW3;
       "PCS_1".wMod4Warn4 := #wMW4;
   END_IF;
END_REGION

REGION Network 16: Module 5 Warnings
   RUNG wire#powerrail
      { S7_Templates := "SrcType := Int" } EQ_Contact(in1 := "PCS_1".iModWarn, in2 := 5)
      wire#w1
      Move(in := #wMW1, out1 => "PCS_1".wMod5Warn1)
      Move(in := #wMW2, out1 => "PCS_1".wMod5Warn2)
   END_RUNG
   RUNG wire#w1
      Move(in := #wMW3, out1 => "PCS_1".wMod5Warn3)
      Move(in := #wMW4, out1 => "PCS_1".wMod5Warn4)
   END_RUNG
   // the same network as SCL:
   IF "PCS_1".iModWarn = 5 THEN
       "PCS_1".wMod5Warn1 := #wMW1;
       "PCS_1".wMod5Warn2 := #wMW2;
       "PCS_1".wMod5Warn3 := #wMW3;
       "PCS_1".wMod5Warn4 := #wMW4;
   END_IF;
END_REGION

REGION Network 17: Module 6 Warnings
   RUNG wire#powerrail
      { S7_Templates := "SrcType := Int" } EQ_Contact(in1 := "PCS_1".iModWarn, in2 := 6)
      wire#w1
      Move(in := #wMW1, out1 => "PCS_1".wMod6Warn1)
      Move(in := #wMW2, out1 => "PCS_1".wMod6Warn2)
   END_RUNG
   RUNG wire#w1
      Move(in := #wMW3, out1 => "PCS_1".wMod6Warn3)
      Move(in := #wMW4, out1 => "PCS_1".wMod6Warn4)
   END_RUNG
   // the same network as SCL:
   IF "PCS_1".iModWarn = 6 THEN
       "PCS_1".wMod6Warn1 := #wMW1;
       "PCS_1".wMod6Warn2 := #wMW2;
       "PCS_1".wMod6Warn3 := #wMW3;
       "PCS_1".wMod6Warn4 := #wMW4;
   END_IF;
END_REGION

REGION Network 19: Fault Modbus Communication
   RUNG wire#powerrail
      Contact( "MbPCS_1-R_slow".ERROR )
      wire#w1
      Coil( "PCS_1".xCommFltSt )
   END_RUNG
   RUNG wire#powerrail
      Contact( "MbPCS_1-R_fast".ERROR )
   END_RUNG wire#w1
   RUNG wire#powerrail
      Contact( "MbPCS_1-W_fast".ERROR )
   END_RUNG wire#w1
   RUNG wire#powerrail
      Contact( "MbPCS_1-W_slow".ERROR )
   END_RUNG wire#w1
   RUNG wire#powerrail
      Contact( "MbMVSKID_1".ERROR )
      Contact( "Reminder".x1 )
      I_Contact( true )
   END_RUNG wire#w1
   // the same network as SCL:
   "PCS_1".xCommFltSt := "MbPCS_1-R_slow".ERROR OR "MbPCS_1-R_fast".ERROR OR "MbPCS_1-W_fast".ERROR OR "MbPCS_1-W_slow".ERROR OR ("MbMVSKID_1".ERROR AND "Reminder".x1 AND NOT true);
END_REGION

REGION Network 20: Inverter Fault
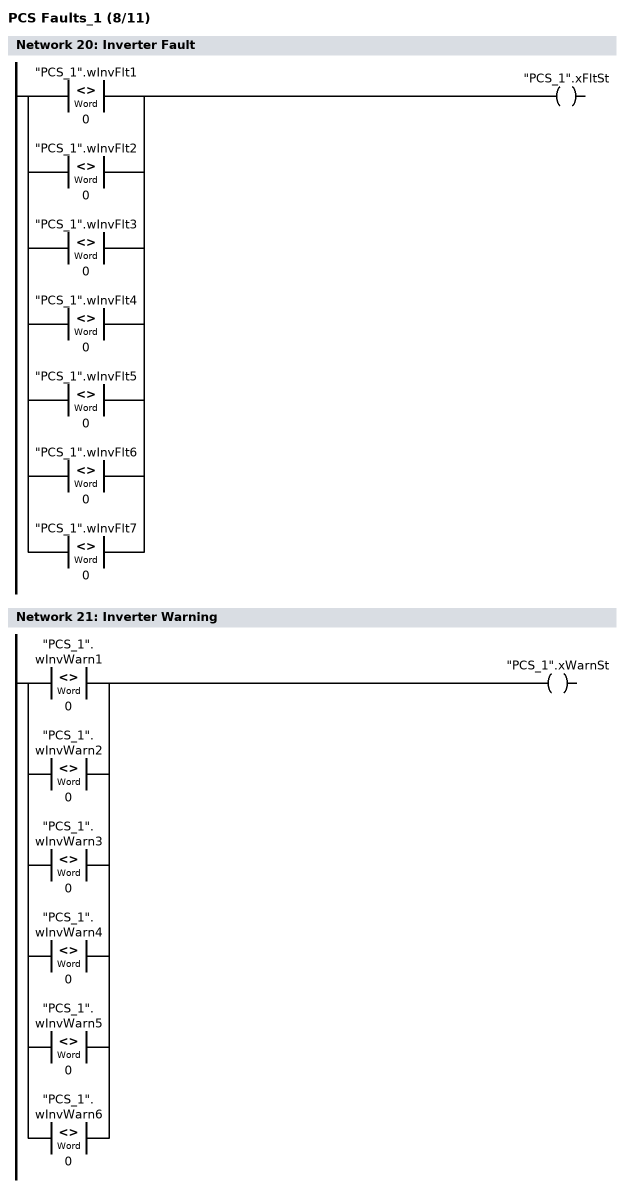
   RUNG wire#powerrail
      { S7_Templates := "SrcType := Word" } NE_Contact(in1 := "PCS_1".wInvFlt1, in2 := 0)
      wire#w1
      Coil( "PCS_1".xFltSt )
   END_RUNG
   RUNG wire#powerrail
      { S7_Templates := "SrcType := Word" } NE_Contact(in1 := "PCS_1".wInvFlt2, in2 := 0)
   END_RUNG wire#w1
   RUNG wire#powerrail
      { S7_Templates := "SrcType := Word" } NE_Contact(in1 := "PCS_1".wInvFlt3, in2 := 0)
   END_RUNG wire#w1
   RUNG wire#powerrail
      { S7_Templates := "SrcType := Word" } NE_Contact(in1 := "PCS_1".wInvFlt4, in2 := 0)
   END_RUNG wire#w1
   RUNG wire#powerrail
      { S7_Templates := "SrcType := Word" } NE_Contact(in1 := "PCS_1".wInvFlt5, in2 := 0)
   END_RUNG wire#w1
   RUNG wire#powerrail
      { S7_Templates := "SrcType := Word" } NE_Contact(in1 := "PCS_1".wInvFlt6, in2 := 0)
   END_RUNG wire#w1
   RUNG wire#powerrail
      { S7_Templates := "SrcType := Word" } NE_Contact(in1 := "PCS_1".wInvFlt7, in2 := 0)
   END_RUNG wire#w1
   // the same network as SCL:
   "PCS_1".xFltSt := ("PCS_1".wInvFlt1 <> 0) OR ("PCS_1".wInvFlt2 <> 0) OR ("PCS_1".wInvFlt3 <> 0) OR ("PCS_1".wInvFlt4 <> 0) OR ("PCS_1".wInvFlt5 <> 0) OR ("PCS_1".wInvFlt6 <> 0) OR ("PCS_1".wInvFlt7 <> 0);
END_REGION

REGION Network 21: Inverter Warning
   RUNG wire#powerrail
      { S7_Templates := "SrcType := Word" } NE_Contact(in1 := "PCS_1".wInvWarn1, in2 := 0)
      wire#w1
      Coil( "PCS_1".xWarnSt )
   END_RUNG
   RUNG wire#powerrail
      { S7_Templates := "SrcType := Word" } NE_Contact(in1 := "PCS_1".wInvWarn2, in2 := 0)
   END_RUNG wire#w1
   RUNG wire#powerrail
      { S7_Templates := "SrcType := Word" } NE_Contact(in1 := "PCS_1".wInvWarn3, in2 := 0)
   END_RUNG wire#w1
   RUNG wire#powerrail
      { S7_Templates := "SrcType := Word" } NE_Contact(in1 := "PCS_1".wInvWarn4, in2 := 0)
   END_RUNG wire#w1
   RUNG wire#powerrail
      { S7_Templates := "SrcType := Word" } NE_Contact(in1 := "PCS_1".wInvWarn5, in2 := 0)
   END_RUNG wire#w1
   RUNG wire#powerrail
      { S7_Templates := "SrcType := Word" } NE_Contact(in1 := "PCS_1".wInvWarn6, in2 := 0)
   END_RUNG wire#w1
   // the same network as SCL:
   "PCS_1".xWarnSt := ("PCS_1".wInvWarn1 <> 0) OR ("PCS_1".wInvWarn2 <> 0) OR ("PCS_1".wInvWarn3 <> 0) OR ("PCS_1".wInvWarn4 <> 0) OR ("PCS_1".wInvWarn5 <> 0) OR ("PCS_1".wInvWarn6 <> 0);
END_REGION

REGION Network 22: Da qua in poi è da chiarire se ci sono warninig e fault relativi ai moduli
END_REGION

REGION Network 23: Bus 1 Mod Fault
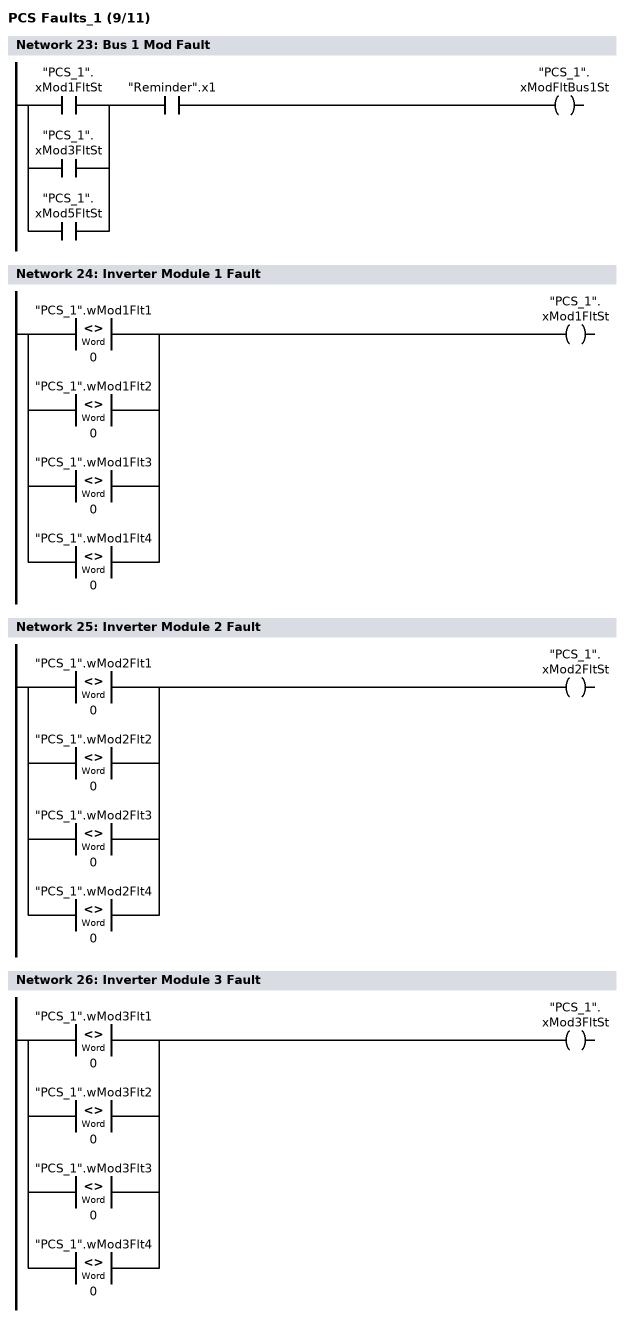
   RUNG wire#powerrail
      Contact( "PCS_1".xMod1FltSt )
      wire#w1
      Contact( "Reminder".x1 )
      Coil( "PCS_1".xModFltBus1St )
   END_RUNG
   RUNG wire#powerrail
      Contact( "PCS_1".xMod3FltSt )
   END_RUNG wire#w1
   RUNG wire#powerrail
      Contact( "PCS_1".xMod5FltSt )
   END_RUNG wire#w1
   // the same network as SCL:
   "PCS_1".xModFltBus1St := ("PCS_1".xMod1FltSt OR "PCS_1".xMod3FltSt OR "PCS_1".xMod5FltSt) AND "Reminder".x1;
END_REGION

REGION Network 24: Inverter Module 1 Fault
   RUNG wire#powerrail
      { S7_Templates := "SrcType := Word" } NE_Contact(in1 := "PCS_1".wMod1Flt1, in2 := 0)
      wire#w1
      Coil( "PCS_1".xMod1FltSt )
   END_RUNG
   RUNG wire#powerrail
      { S7_Templates := "SrcType := Word" } NE_Contact(in1 := "PCS_1".wMod1Flt2, in2 := 0)
   END_RUNG wire#w1
   RUNG wire#powerrail
      { S7_Templates := "SrcType := Word" } NE_Contact(in1 := "PCS_1".wMod1Flt3, in2 := 0)
   END_RUNG wire#w1
   RUNG wire#powerrail
      { S7_Templates := "SrcType := Word" } NE_Contact(in1 := "PCS_1".wMod1Flt4, in2 := 0)
   END_RUNG wire#w1
   // the same network as SCL:
   "PCS_1".xMod1FltSt := ("PCS_1".wMod1Flt1 <> 0) OR ("PCS_1".wMod1Flt2 <> 0) OR ("PCS_1".wMod1Flt3 <> 0) OR ("PCS_1".wMod1Flt4 <> 0);
END_REGION

REGION Network 25: Inverter Module 2 Fault
   RUNG wire#powerrail
      { S7_Templates := "SrcType := Word" } NE_Contact(in1 := "PCS_1".wMod2Flt1, in2 := 0)
      wire#w1
      Coil( "PCS_1".xMod2FltSt )
   END_RUNG
   RUNG wire#powerrail
      { S7_Templates := "SrcType := Word" } NE_Contact(in1 := "PCS_1".wMod2Flt2, in2 := 0)
   END_RUNG wire#w1
   RUNG wire#powerrail
      { S7_Templates := "SrcType := Word" } NE_Contact(in1 := "PCS_1".wMod2Flt3, in2 := 0)
   END_RUNG wire#w1
   RUNG wire#powerrail
      { S7_Templates := "SrcType := Word" } NE_Contact(in1 := "PCS_1".wMod2Flt4, in2 := 0)
   END_RUNG wire#w1
   // the same network as SCL:
   "PCS_1".xMod2FltSt := ("PCS_1".wMod2Flt1 <> 0) OR ("PCS_1".wMod2Flt2 <> 0) OR ("PCS_1".wMod2Flt3 <> 0) OR ("PCS_1".wMod2Flt4 <> 0);
END_REGION

REGION Network 26: Inverter Module 3 Fault
   RUNG wire#powerrail
      { S7_Templates := "SrcType := Word" } NE_Contact(in1 := "PCS_1".wMod3Flt1, in2 := 0)
      wire#w1
      Coil( "PCS_1".xMod3FltSt )
   END_RUNG
   RUNG wire#powerrail
      { S7_Templates := "SrcType := Word" } NE_Contact(in1 := "PCS_1".wMod3Flt2, in2 := 0)
   END_RUNG wire#w1
   RUNG wire#powerrail
      { S7_Templates := "SrcType := Word" } NE_Contact(in1 := "PCS_1".wMod3Flt3, in2 := 0)
   END_RUNG wire#w1
   RUNG wire#powerrail
      { S7_Templates := "SrcType := Word" } NE_Contact(in1 := "PCS_1".wMod3Flt4, in2 := 0)
   END_RUNG wire#w1
   // the same network as SCL:
   "PCS_1".xMod3FltSt := ("PCS_1".wMod3Flt1 <> 0) OR ("PCS_1".wMod3Flt2 <> 0) OR ("PCS_1".wMod3Flt3 <> 0) OR ("PCS_1".wMod3Flt4 <> 0);
END_REGION

REGION Network 27: Inverter Module 4 Fault
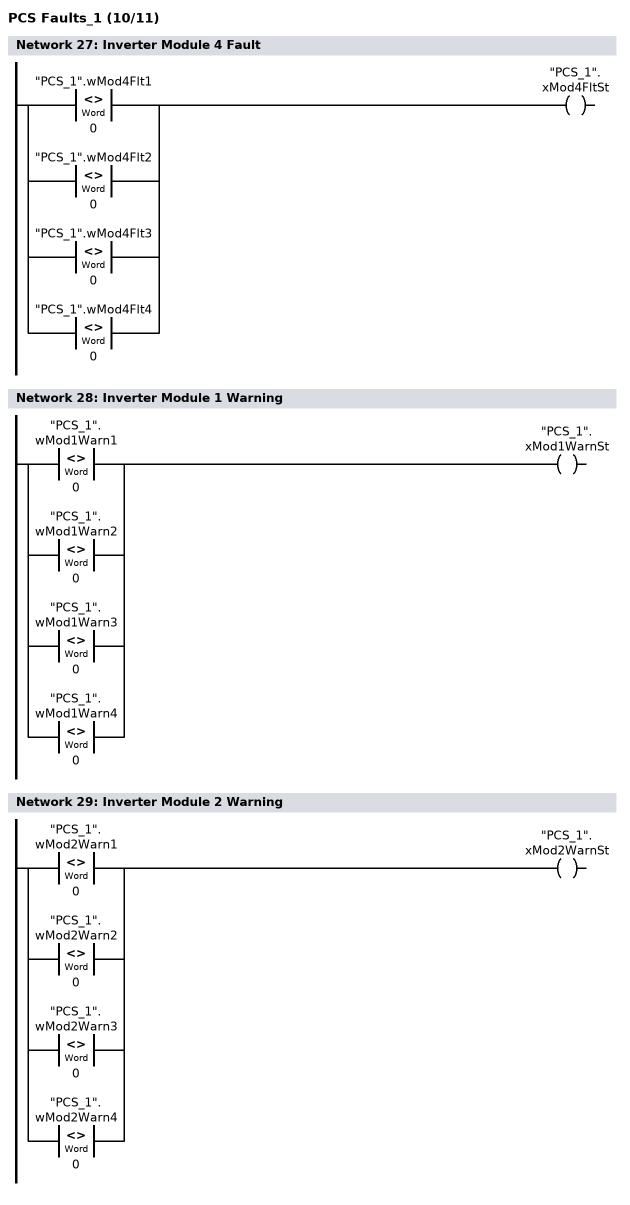
   RUNG wire#powerrail
      { S7_Templates := "SrcType := Word" } NE_Contact(in1 := "PCS_1".wMod4Flt1, in2 := 0)
      wire#w1
      Coil( "PCS_1".xMod4FltSt )
   END_RUNG
   RUNG wire#powerrail
      { S7_Templates := "SrcType := Word" } NE_Contact(in1 := "PCS_1".wMod4Flt2, in2 := 0)
   END_RUNG wire#w1
   RUNG wire#powerrail
      { S7_Templates := "SrcType := Word" } NE_Contact(in1 := "PCS_1".wMod4Flt3, in2 := 0)
   END_RUNG wire#w1
   RUNG wire#powerrail
      { S7_Templates := "SrcType := Word" } NE_Contact(in1 := "PCS_1".wMod4Flt4, in2 := 0)
   END_RUNG wire#w1
   // the same network as SCL:
   "PCS_1".xMod4FltSt := ("PCS_1".wMod4Flt1 <> 0) OR ("PCS_1".wMod4Flt2 <> 0) OR ("PCS_1".wMod4Flt3 <> 0) OR ("PCS_1".wMod4Flt4 <> 0);
END_REGION

REGION Network 28: Inverter Module 1 Warning
   RUNG wire#powerrail
      { S7_Templates := "SrcType := Word" } NE_Contact(in1 := "PCS_1".wMod1Warn1, in2 := 0)
      wire#w1
      Coil( "PCS_1".xMod1WarnSt )
   END_RUNG
   RUNG wire#powerrail
      { S7_Templates := "SrcType := Word" } NE_Contact(in1 := "PCS_1".wMod1Warn2, in2 := 0)
   END_RUNG wire#w1
   RUNG wire#powerrail
      { S7_Templates := "SrcType := Word" } NE_Contact(in1 := "PCS_1".wMod1Warn3, in2 := 0)
   END_RUNG wire#w1
   RUNG wire#powerrail
      { S7_Templates := "SrcType := Word" } NE_Contact(in1 := "PCS_1".wMod1Warn4, in2 := 0)
   END_RUNG wire#w1
   // the same network as SCL:
   "PCS_1".xMod1WarnSt := ("PCS_1".wMod1Warn1 <> 0) OR ("PCS_1".wMod1Warn2 <> 0) OR ("PCS_1".wMod1Warn3 <> 0) OR ("PCS_1".wMod1Warn4 <> 0);
END_REGION

REGION Network 29: Inverter Module 2 Warning
   RUNG wire#powerrail
      { S7_Templates := "SrcType := Word" } NE_Contact(in1 := "PCS_1".wMod2Warn1, in2 := 0)
      wire#w1
      Coil( "PCS_1".xMod2WarnSt )
   END_RUNG
   RUNG wire#powerrail
      { S7_Templates := "SrcType := Word" } NE_Contact(in1 := "PCS_1".wMod2Warn2, in2 := 0)
   END_RUNG wire#w1
   RUNG wire#powerrail
      { S7_Templates := "SrcType := Word" } NE_Contact(in1 := "PCS_1".wMod2Warn3, in2 := 0)
   END_RUNG wire#w1
   RUNG wire#powerrail
      { S7_Templates := "SrcType := Word" } NE_Contact(in1 := "PCS_1".wMod2Warn4, in2 := 0)
   END_RUNG wire#w1
   // the same network as SCL:
   "PCS_1".xMod2WarnSt := ("PCS_1".wMod2Warn1 <> 0) OR ("PCS_1".wMod2Warn2 <> 0) OR ("PCS_1".wMod2Warn3 <> 0) OR ("PCS_1".wMod2Warn4 <> 0);
END_REGION

REGION Network 30: Inverter Module 3 Warning
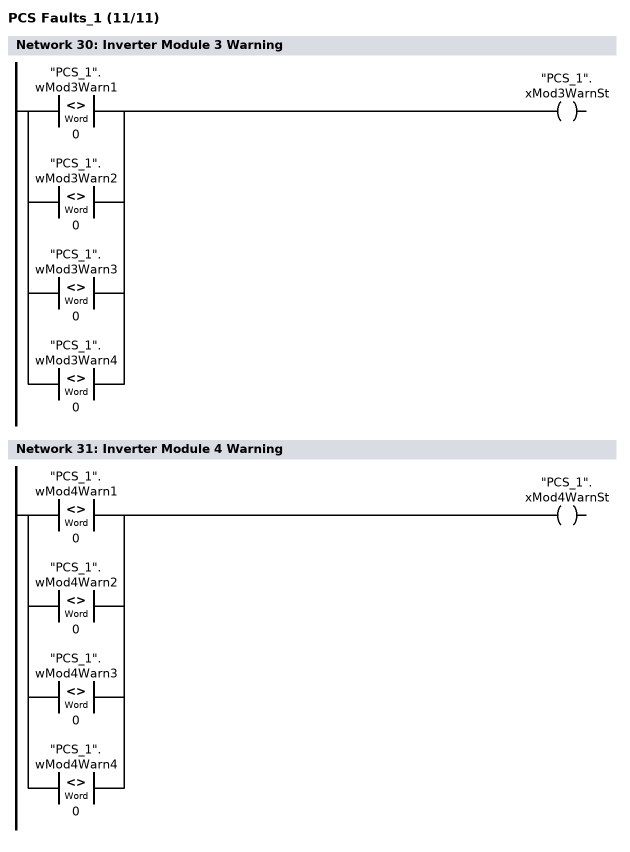
   RUNG wire#powerrail
      { S7_Templates := "SrcType := Word" } NE_Contact(in1 := "PCS_1".wMod3Warn1, in2 := 0)
      wire#w1
      Coil( "PCS_1".xMod3WarnSt )
   END_RUNG
   RUNG wire#powerrail
      { S7_Templates := "SrcType := Word" } NE_Contact(in1 := "PCS_1".wMod3Warn2, in2 := 0)
   END_RUNG wire#w1
   RUNG wire#powerrail
      { S7_Templates := "SrcType := Word" } NE_Contact(in1 := "PCS_1".wMod3Warn3, in2 := 0)
   END_RUNG wire#w1
   RUNG wire#powerrail
      { S7_Templates := "SrcType := Word" } NE_Contact(in1 := "PCS_1".wMod3Warn4, in2 := 0)
   END_RUNG wire#w1
   // the same network as SCL:
   "PCS_1".xMod3WarnSt := ("PCS_1".wMod3Warn1 <> 0) OR ("PCS_1".wMod3Warn2 <> 0) OR ("PCS_1".wMod3Warn3 <> 0) OR ("PCS_1".wMod3Warn4 <> 0);
END_REGION

REGION Network 31: Inverter Module 4 Warning
   RUNG wire#powerrail
      { S7_Templates := "SrcType := Word" } NE_Contact(in1 := "PCS_1".wMod4Warn1, in2 := 0)
      wire#w1
      Coil( "PCS_1".xMod4WarnSt )
   END_RUNG
   RUNG wire#powerrail
      { S7_Templates := "SrcType := Word" } NE_Contact(in1 := "PCS_1".wMod4Warn2, in2 := 0)
   END_RUNG wire#w1
   RUNG wire#powerrail
      { S7_Templates := "SrcType := Word" } NE_Contact(in1 := "PCS_1".wMod4Warn3, in2 := 0)
   END_RUNG wire#w1
   RUNG wire#powerrail
      { S7_Templates := "SrcType := Word" } NE_Contact(in1 := "PCS_1".wMod4Warn4, in2 := 0)
   END_RUNG wire#w1
   // the same network as SCL:
   "PCS_1".xMod4WarnSt := ("PCS_1".wMod4Warn1 <> 0) OR ("PCS_1".wMod4Warn2 <> 0) OR ("PCS_1".wMod4Warn3 <> 0) OR ("PCS_1".wMod4Warn4 <> 0);
END_REGION
END_FUNCTION

FUNCTION "PCS R (F)_1" : Void   // FC47, LAD
TITLE = ModBus TCP for PCS Power Electronics
{ S7_Optimized_Access := 'TRUE' }
VERSION : 0.1
// stored: AutoNumber true, IsIECCheckEnabled false, SetENOAutomatically false, UDAEnableTagReadback false
   VAR_TEMP
      rVac : Real;
   END_VAR
   VAR_TEMP   // added for the SCL form of the ladder/FBD networks
      _w1 : Bool;
   END_VAR
BEGIN

REGION Network 1: Function Modbus Client 10
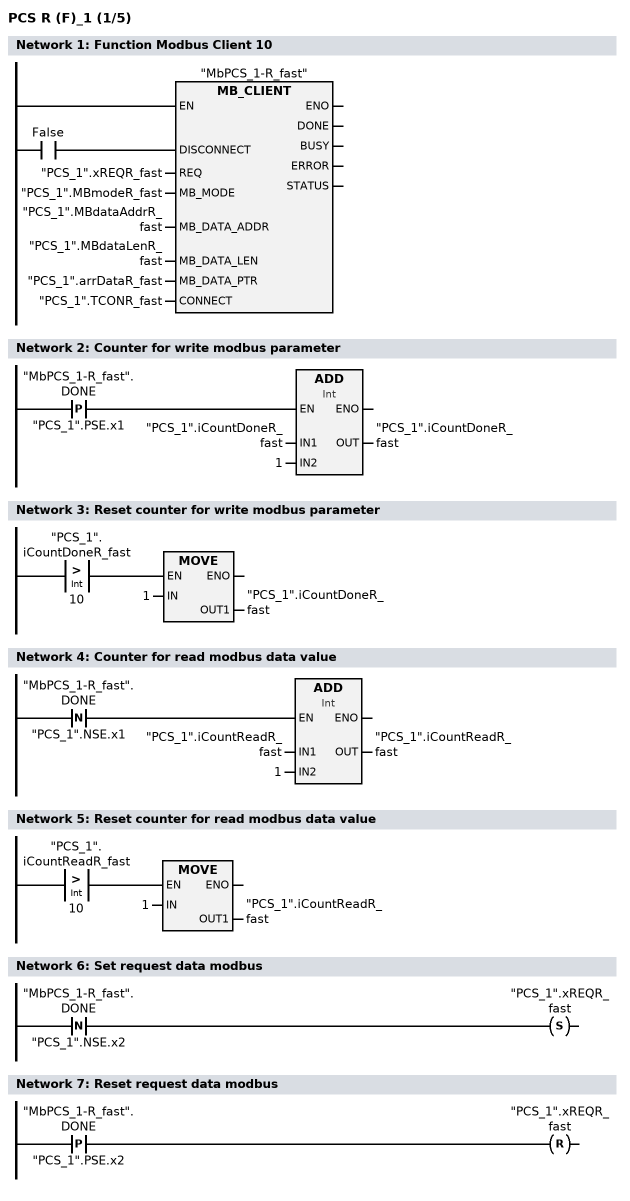
   RUNG wire#powerrail
      "MbPCS_1-R_fast".MB_CLIENT(DISCONNECT := wire#w1, REQ := "PCS_1".xREQR_fast, MB_MODE := "PCS_1".MBmodeR_fast, MB_DATA_ADDR := "PCS_1".MBdataAddrR_fast, MB_DATA_LEN := "PCS_1".MBdataLenR_fast, MB_DATA_PTR := "PCS_1".arrDataR_fast, CONNECT := "PCS_1".TCONR_fast, DONE =>, BUSY =>, ERROR =>, STATUS =>)
   END_RUNG
   RUNG wire#powerrail
      Contact( False )
   END_RUNG wire#w1
   // the same network as SCL:
   "MbPCS_1-R_fast"(DISCONNECT := False,   // MB_CLIENT
                    REQ := "PCS_1".xREQR_fast,
                    MB_MODE := "PCS_1".MBmodeR_fast,
                    MB_DATA_ADDR := "PCS_1".MBdataAddrR_fast,
                    MB_DATA_LEN := "PCS_1".MBdataLenR_fast,
                    MB_DATA_PTR := "PCS_1".arrDataR_fast,
                    CONNECT := "PCS_1".TCONR_fast);
END_REGION

REGION Network 2: Counter for write modbus parameter
   RUNG wire#powerrail
      P_Contact(operand := "MbPCS_1-R_fast".DONE, bit := "PCS_1".PSE.x1)
      { S7_Templates := "SrcType := Int" } Add(in1 := "PCS_1".iCountDoneR_fast, in2 := 1, out => "PCS_1".iCountDoneR_fast)
   END_RUNG
   // the same network as SCL:
   #_w1 := "MbPCS_1-R_fast".DONE AND NOT "PCS_1".PSE.x1;   // rising edge of "MbPCS_1-R_fast".DONE
   "PCS_1".PSE.x1 := "MbPCS_1-R_fast".DONE;
   IF #_w1 THEN "PCS_1".iCountDoneR_fast := "PCS_1".iCountDoneR_fast + 1; END_IF;
END_REGION

REGION Network 3: Reset counter for write modbus parameter
   RUNG wire#powerrail
      { S7_Templates := "SrcType := Int" } GT_Contact(in1 := "PCS_1".iCountDoneR_fast, in2 := 10)
      Move(in := 1, out1 => "PCS_1".iCountDoneR_fast)
   END_RUNG
   // the same network as SCL:
   IF "PCS_1".iCountDoneR_fast > 10 THEN "PCS_1".iCountDoneR_fast := 1; END_IF;
END_REGION

REGION Network 4: Counter for read modbus data value
   RUNG wire#powerrail
      N_Contact(operand := "MbPCS_1-R_fast".DONE, bit := "PCS_1".NSE.x1)
      { S7_Templates := "SrcType := Int" } Add(in1 := "PCS_1".iCountReadR_fast, in2 := 1, out => "PCS_1".iCountReadR_fast)
   END_RUNG
   // the same network as SCL:
   #_w1 := NOT "MbPCS_1-R_fast".DONE AND "PCS_1".NSE.x1;   // falling edge of "MbPCS_1-R_fast".DONE
   "PCS_1".NSE.x1 := "MbPCS_1-R_fast".DONE;
   IF #_w1 THEN "PCS_1".iCountReadR_fast := "PCS_1".iCountReadR_fast + 1; END_IF;
END_REGION

REGION Network 5: Reset counter for read modbus data value
   RUNG wire#powerrail
      { S7_Templates := "SrcType := Int" } GT_Contact(in1 := "PCS_1".iCountReadR_fast, in2 := 10)
      Move(in := 1, out1 => "PCS_1".iCountReadR_fast)
   END_RUNG
   // the same network as SCL:
   IF "PCS_1".iCountReadR_fast > 10 THEN "PCS_1".iCountReadR_fast := 1; END_IF;
END_REGION

REGION Network 6: Set request data modbus
   RUNG wire#powerrail
      N_Contact(operand := "MbPCS_1-R_fast".DONE, bit := "PCS_1".NSE.x2)
      S_Coil( "PCS_1".xREQR_fast )
   END_RUNG
   // the same network as SCL:
   #_w1 := NOT "MbPCS_1-R_fast".DONE AND "PCS_1".NSE.x2;   // falling edge of "MbPCS_1-R_fast".DONE
   "PCS_1".NSE.x2 := "MbPCS_1-R_fast".DONE;
   IF #_w1 THEN "PCS_1".xREQR_fast := TRUE; END_IF;
END_REGION

REGION Network 7: Reset request data modbus
   RUNG wire#powerrail
      P_Contact(operand := "MbPCS_1-R_fast".DONE, bit := "PCS_1".PSE.x2)
      R_Coil( "PCS_1".xREQR_fast )
   END_RUNG
   // the same network as SCL:
   #_w1 := "MbPCS_1-R_fast".DONE AND NOT "PCS_1".PSE.x2;   // rising edge of "MbPCS_1-R_fast".DONE
   "PCS_1".PSE.x2 := "MbPCS_1-R_fast".DONE;
   IF #_w1 THEN "PCS_1".xREQR_fast := FALSE; END_IF;
END_REGION

REGION Network 8: Write R_Block1 parameter - new
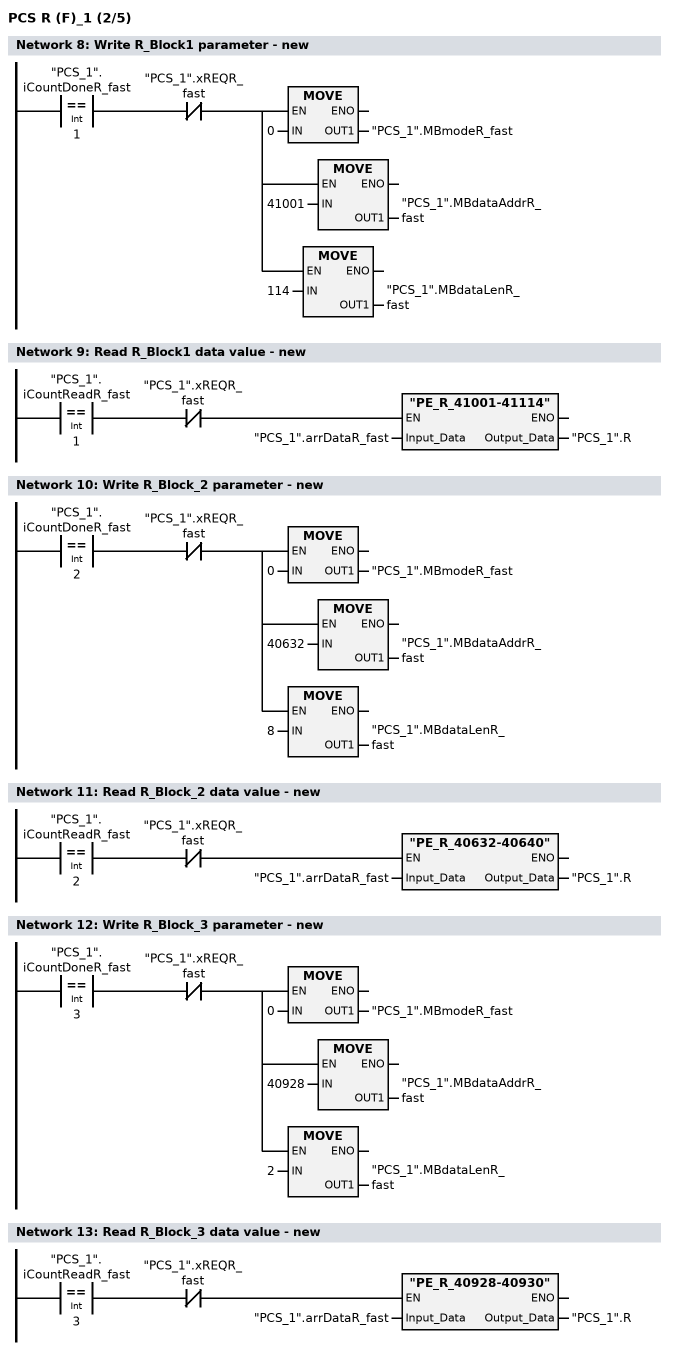
   RUNG wire#powerrail
      { S7_Templates := "SrcType := Int" } EQ_Contact(in1 := "PCS_1".iCountDoneR_fast, in2 := 1)
      I_Contact( "PCS_1".xREQR_fast )
      wire#w1
      Move(in := 0, out1 => "PCS_1".MBmodeR_fast)
   END_RUNG
   RUNG wire#w1
      Move(in := 41001, out1 => "PCS_1".MBdataAddrR_fast)
   END_RUNG
   RUNG wire#w1
      Move(in := 114, out1 => "PCS_1".MBdataLenR_fast)
   END_RUNG
   // the same network as SCL:
   IF ("PCS_1".iCountDoneR_fast = 1) AND NOT "PCS_1".xREQR_fast THEN
       "PCS_1".MBmodeR_fast := 0;
       "PCS_1".MBdataAddrR_fast := 41001;
       "PCS_1".MBdataLenR_fast := 114;
   END_IF;
END_REGION

REGION Network 9: Read R_Block1 data value - new
   RUNG wire#powerrail
      { S7_Templates := "SrcType := Int" } EQ_Contact(in1 := "PCS_1".iCountReadR_fast, in2 := 1)
      I_Contact( "PCS_1".xREQR_fast )
      "PE_R_41001-41114"(Input_Data := "PCS_1".arrDataR_fast, Output_Data => "PCS_1".R)
   END_RUNG
   // the same network as SCL:
   IF ("PCS_1".iCountReadR_fast = 1) AND NOT "PCS_1".xREQR_fast THEN
       "PE_R_41001-41114"(Input_Data := "PCS_1".arrDataR_fast, Output_Data => "PCS_1".R);
   END_IF;
END_REGION

REGION Network 10: Write R_Block_2 parameter - new
   RUNG wire#powerrail
      { S7_Templates := "SrcType := Int" } EQ_Contact(in1 := "PCS_1".iCountDoneR_fast, in2 := 2)
      I_Contact( "PCS_1".xREQR_fast )
      wire#w1
      Move(in := 0, out1 => "PCS_1".MBmodeR_fast)
   END_RUNG
   RUNG wire#w1
      Move(in := 40632, out1 => "PCS_1".MBdataAddrR_fast)
   END_RUNG
   RUNG wire#w1
      Move(in := 8, out1 => "PCS_1".MBdataLenR_fast)
   END_RUNG
   // the same network as SCL:
   IF ("PCS_1".iCountDoneR_fast = 2) AND NOT "PCS_1".xREQR_fast THEN
       "PCS_1".MBmodeR_fast := 0;
       "PCS_1".MBdataAddrR_fast := 40632;
       "PCS_1".MBdataLenR_fast := 8;
   END_IF;
END_REGION

REGION Network 11: Read R_Block_2 data value - new
   RUNG wire#powerrail
      { S7_Templates := "SrcType := Int" } EQ_Contact(in1 := "PCS_1".iCountReadR_fast, in2 := 2)
      I_Contact( "PCS_1".xREQR_fast )
      "PE_R_40632-40640"(Input_Data := "PCS_1".arrDataR_fast, Output_Data => "PCS_1".R)
   END_RUNG
   // the same network as SCL:
   IF ("PCS_1".iCountReadR_fast = 2) AND NOT "PCS_1".xREQR_fast THEN
       "PE_R_40632-40640"(Input_Data := "PCS_1".arrDataR_fast, Output_Data => "PCS_1".R);
   END_IF;
END_REGION

REGION Network 12: Write R_Block_3 parameter - new
   RUNG wire#powerrail
      { S7_Templates := "SrcType := Int" } EQ_Contact(in1 := "PCS_1".iCountDoneR_fast, in2 := 3)
      I_Contact( "PCS_1".xREQR_fast )
      wire#w1
      Move(in := 0, out1 => "PCS_1".MBmodeR_fast)
   END_RUNG
   RUNG wire#w1
      Move(in := 40928, out1 => "PCS_1".MBdataAddrR_fast)
   END_RUNG
   RUNG wire#w1
      Move(in := 2, out1 => "PCS_1".MBdataLenR_fast)
   END_RUNG
   // the same network as SCL:
   IF ("PCS_1".iCountDoneR_fast = 3) AND NOT "PCS_1".xREQR_fast THEN
       "PCS_1".MBmodeR_fast := 0;
       "PCS_1".MBdataAddrR_fast := 40928;
       "PCS_1".MBdataLenR_fast := 2;
   END_IF;
END_REGION

REGION Network 13: Read R_Block_3 data value - new
   RUNG wire#powerrail
      { S7_Templates := "SrcType := Int" } EQ_Contact(in1 := "PCS_1".iCountReadR_fast, in2 := 3)
      I_Contact( "PCS_1".xREQR_fast )
      "PE_R_40928-40930"(Input_Data := "PCS_1".arrDataR_fast, Output_Data => "PCS_1".R)
   END_RUNG
   // the same network as SCL:
   IF ("PCS_1".iCountReadR_fast = 3) AND NOT "PCS_1".xREQR_fast THEN
       "PE_R_40928-40930"(Input_Data := "PCS_1".arrDataR_fast, Output_Data => "PCS_1".R);
   END_IF;
END_REGION

REGION Network 14: Write R_Block_4 parameter - new
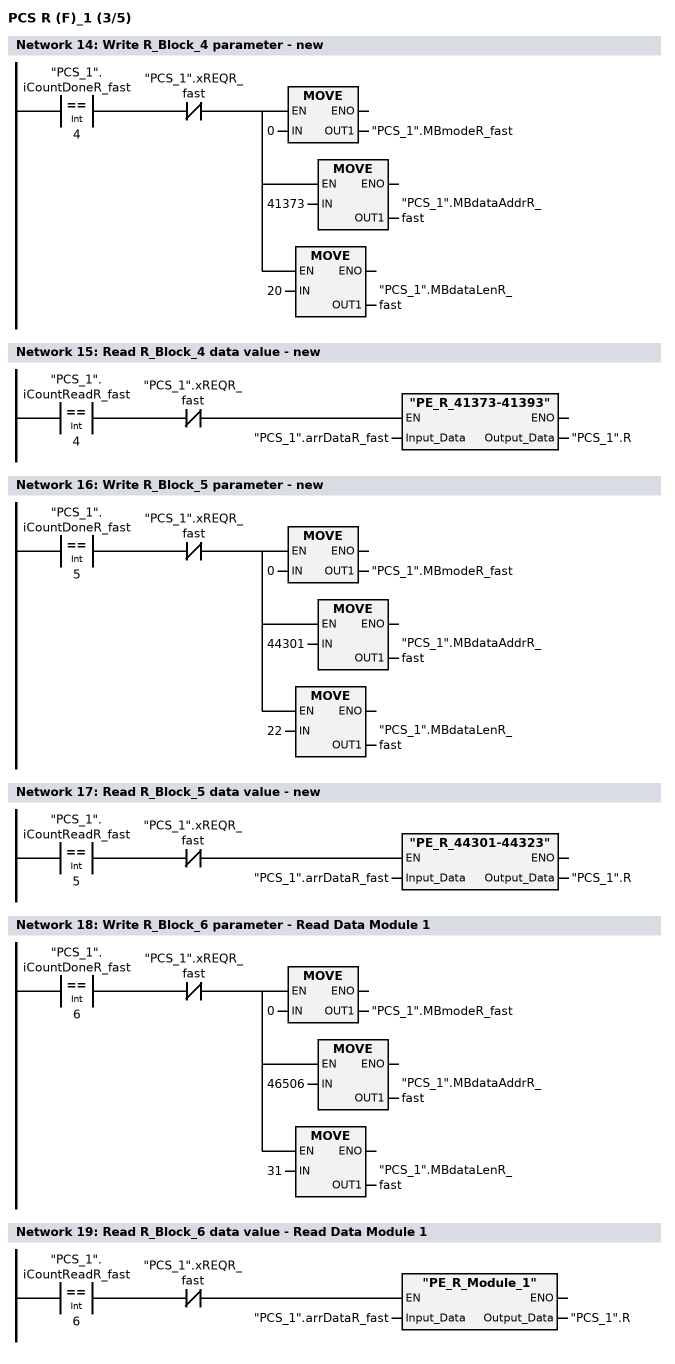
   RUNG wire#powerrail
      { S7_Templates := "SrcType := Int" } EQ_Contact(in1 := "PCS_1".iCountDoneR_fast, in2 := 4)
      I_Contact( "PCS_1".xREQR_fast )
      wire#w1
      Move(in := 0, out1 => "PCS_1".MBmodeR_fast)
   END_RUNG
   RUNG wire#w1
      Move(in := 41373, out1 => "PCS_1".MBdataAddrR_fast)
   END_RUNG
   RUNG wire#w1
      Move(in := 20, out1 => "PCS_1".MBdataLenR_fast)
   END_RUNG
   // the same network as SCL:
   IF ("PCS_1".iCountDoneR_fast = 4) AND NOT "PCS_1".xREQR_fast THEN
       "PCS_1".MBmodeR_fast := 0;
       "PCS_1".MBdataAddrR_fast := 41373;
       "PCS_1".MBdataLenR_fast := 20;
   END_IF;
END_REGION

REGION Network 15: Read R_Block_4 data value - new
   RUNG wire#powerrail
      { S7_Templates := "SrcType := Int" } EQ_Contact(in1 := "PCS_1".iCountReadR_fast, in2 := 4)
      I_Contact( "PCS_1".xREQR_fast )
      "PE_R_41373-41393"(Input_Data := "PCS_1".arrDataR_fast, Output_Data => "PCS_1".R)
   END_RUNG
   // the same network as SCL:
   IF ("PCS_1".iCountReadR_fast = 4) AND NOT "PCS_1".xREQR_fast THEN
       "PE_R_41373-41393"(Input_Data := "PCS_1".arrDataR_fast, Output_Data => "PCS_1".R);
   END_IF;
END_REGION

REGION Network 16: Write R_Block_5 parameter - new
   RUNG wire#powerrail
      { S7_Templates := "SrcType := Int" } EQ_Contact(in1 := "PCS_1".iCountDoneR_fast, in2 := 5)
      I_Contact( "PCS_1".xREQR_fast )
      wire#w1
      Move(in := 0, out1 => "PCS_1".MBmodeR_fast)
   END_RUNG
   RUNG wire#w1
      Move(in := 44301, out1 => "PCS_1".MBdataAddrR_fast)
   END_RUNG
   RUNG wire#w1
      Move(in := 22, out1 => "PCS_1".MBdataLenR_fast)
   END_RUNG
   // the same network as SCL:
   IF ("PCS_1".iCountDoneR_fast = 5) AND NOT "PCS_1".xREQR_fast THEN
       "PCS_1".MBmodeR_fast := 0;
       "PCS_1".MBdataAddrR_fast := 44301;
       "PCS_1".MBdataLenR_fast := 22;
   END_IF;
END_REGION

REGION Network 17: Read R_Block_5 data value - new
   RUNG wire#powerrail
      { S7_Templates := "SrcType := Int" } EQ_Contact(in1 := "PCS_1".iCountReadR_fast, in2 := 5)
      I_Contact( "PCS_1".xREQR_fast )
      "PE_R_44301-44323"(Input_Data := "PCS_1".arrDataR_fast, Output_Data => "PCS_1".R)
   END_RUNG
   // the same network as SCL:
   IF ("PCS_1".iCountReadR_fast = 5) AND NOT "PCS_1".xREQR_fast THEN
       "PE_R_44301-44323"(Input_Data := "PCS_1".arrDataR_fast, Output_Data => "PCS_1".R);
   END_IF;
END_REGION

REGION Network 18: Write R_Block_6 parameter - Read Data Module 1
   RUNG wire#powerrail
      { S7_Templates := "SrcType := Int" } EQ_Contact(in1 := "PCS_1".iCountDoneR_fast, in2 := 6)
      I_Contact( "PCS_1".xREQR_fast )
      wire#w1
      Move(in := 0, out1 => "PCS_1".MBmodeR_fast)
   END_RUNG
   RUNG wire#w1
      Move(in := 46506, out1 => "PCS_1".MBdataAddrR_fast)
   END_RUNG
   RUNG wire#w1
      Move(in := 31, out1 => "PCS_1".MBdataLenR_fast)
   END_RUNG
   // the same network as SCL:
   IF ("PCS_1".iCountDoneR_fast = 6) AND NOT "PCS_1".xREQR_fast THEN
       "PCS_1".MBmodeR_fast := 0;
       "PCS_1".MBdataAddrR_fast := 46506;
       "PCS_1".MBdataLenR_fast := 31;
   END_IF;
END_REGION

REGION Network 19: Read R_Block_6 data value - Read Data Module 1
   RUNG wire#powerrail
      { S7_Templates := "SrcType := Int" } EQ_Contact(in1 := "PCS_1".iCountReadR_fast, in2 := 6)
      I_Contact( "PCS_1".xREQR_fast )
      "PE_R_Module_1"(Input_Data := "PCS_1".arrDataR_fast, Output_Data => "PCS_1".R)
   END_RUNG
   // the same network as SCL:
   IF ("PCS_1".iCountReadR_fast = 6) AND NOT "PCS_1".xREQR_fast THEN
       "PE_R_Module_1"(Input_Data := "PCS_1".arrDataR_fast, Output_Data => "PCS_1".R);
   END_IF;
END_REGION

REGION Network 20: Write R_Block_7 parameter - Read Data Module 2
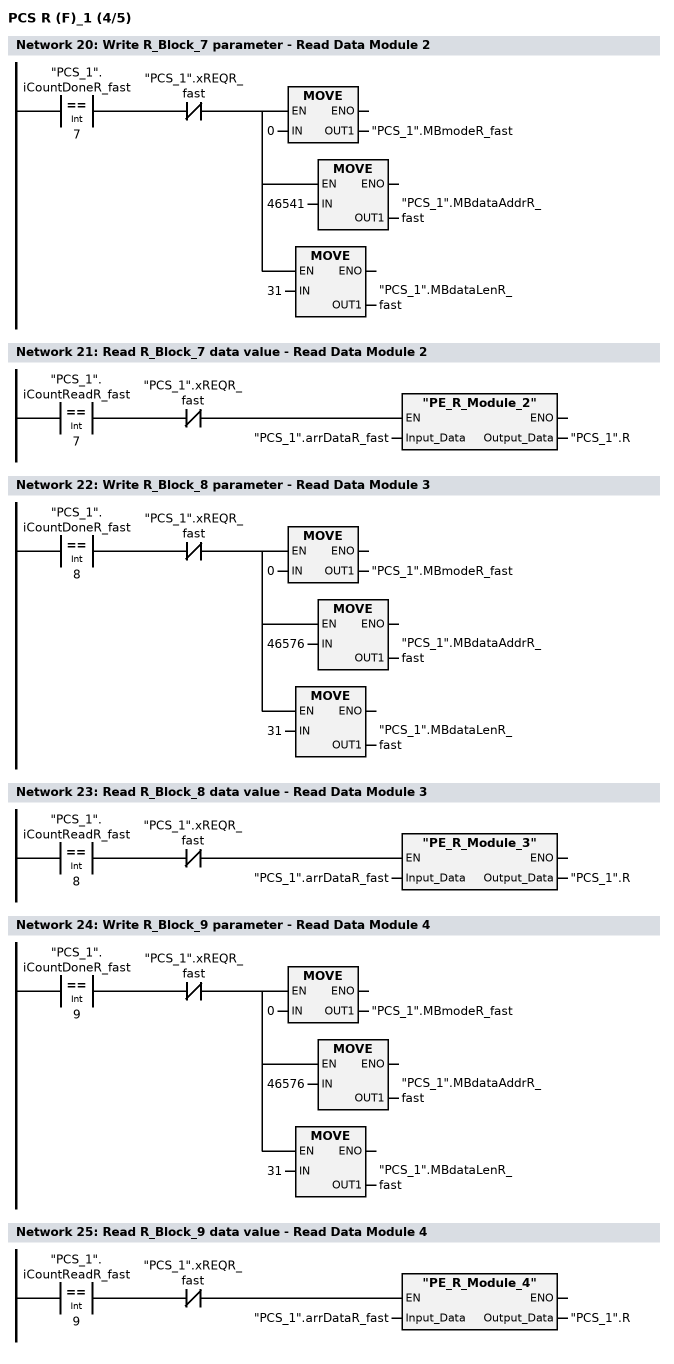
   RUNG wire#powerrail
      { S7_Templates := "SrcType := Int" } EQ_Contact(in1 := "PCS_1".iCountDoneR_fast, in2 := 7)
      I_Contact( "PCS_1".xREQR_fast )
      wire#w1
      Move(in := 0, out1 => "PCS_1".MBmodeR_fast)
   END_RUNG
   RUNG wire#w1
      Move(in := 46541, out1 => "PCS_1".MBdataAddrR_fast)
   END_RUNG
   RUNG wire#w1
      Move(in := 31, out1 => "PCS_1".MBdataLenR_fast)
   END_RUNG
   // the same network as SCL:
   IF ("PCS_1".iCountDoneR_fast = 7) AND NOT "PCS_1".xREQR_fast THEN
       "PCS_1".MBmodeR_fast := 0;
       "PCS_1".MBdataAddrR_fast := 46541;
       "PCS_1".MBdataLenR_fast := 31;
   END_IF;
END_REGION

REGION Network 21: Read R_Block_7 data value - Read Data Module 2
   RUNG wire#powerrail
      { S7_Templates := "SrcType := Int" } EQ_Contact(in1 := "PCS_1".iCountReadR_fast, in2 := 7)
      I_Contact( "PCS_1".xREQR_fast )
      "PE_R_Module_2"(Input_Data := "PCS_1".arrDataR_fast, Output_Data => "PCS_1".R)
   END_RUNG
   // the same network as SCL:
   IF ("PCS_1".iCountReadR_fast = 7) AND NOT "PCS_1".xREQR_fast THEN
       "PE_R_Module_2"(Input_Data := "PCS_1".arrDataR_fast, Output_Data => "PCS_1".R);
   END_IF;
END_REGION

REGION Network 22: Write R_Block_8 parameter - Read Data Module 3
   RUNG wire#powerrail
      { S7_Templates := "SrcType := Int" } EQ_Contact(in1 := "PCS_1".iCountDoneR_fast, in2 := 8)
      I_Contact( "PCS_1".xREQR_fast )
      wire#w1
      Move(in := 0, out1 => "PCS_1".MBmodeR_fast)
   END_RUNG
   RUNG wire#w1
      Move(in := 46576, out1 => "PCS_1".MBdataAddrR_fast)
   END_RUNG
   RUNG wire#w1
      Move(in := 31, out1 => "PCS_1".MBdataLenR_fast)
   END_RUNG
   // the same network as SCL:
   IF ("PCS_1".iCountDoneR_fast = 8) AND NOT "PCS_1".xREQR_fast THEN
       "PCS_1".MBmodeR_fast := 0;
       "PCS_1".MBdataAddrR_fast := 46576;
       "PCS_1".MBdataLenR_fast := 31;
   END_IF;
END_REGION

REGION Network 23: Read R_Block_8 data value - Read Data Module 3
   RUNG wire#powerrail
      { S7_Templates := "SrcType := Int" } EQ_Contact(in1 := "PCS_1".iCountReadR_fast, in2 := 8)
      I_Contact( "PCS_1".xREQR_fast )
      "PE_R_Module_3"(Input_Data := "PCS_1".arrDataR_fast, Output_Data => "PCS_1".R)
   END_RUNG
   // the same network as SCL:
   IF ("PCS_1".iCountReadR_fast = 8) AND NOT "PCS_1".xREQR_fast THEN
       "PE_R_Module_3"(Input_Data := "PCS_1".arrDataR_fast, Output_Data => "PCS_1".R);
   END_IF;
END_REGION

REGION Network 24: Write R_Block_9 parameter - Read Data Module 4
   RUNG wire#powerrail
      { S7_Templates := "SrcType := Int" } EQ_Contact(in1 := "PCS_1".iCountDoneR_fast, in2 := 9)
      I_Contact( "PCS_1".xREQR_fast )
      wire#w1
      Move(in := 0, out1 => "PCS_1".MBmodeR_fast)
   END_RUNG
   RUNG wire#w1
      Move(in := 46576, out1 => "PCS_1".MBdataAddrR_fast)
   END_RUNG
   RUNG wire#w1
      Move(in := 31, out1 => "PCS_1".MBdataLenR_fast)
   END_RUNG
   // the same network as SCL:
   IF ("PCS_1".iCountDoneR_fast = 9) AND NOT "PCS_1".xREQR_fast THEN
       "PCS_1".MBmodeR_fast := 0;
       "PCS_1".MBdataAddrR_fast := 46576;
       "PCS_1".MBdataLenR_fast := 31;
   END_IF;
END_REGION

REGION Network 25: Read R_Block_9 data value - Read Data Module 4
   RUNG wire#powerrail
      { S7_Templates := "SrcType := Int" } EQ_Contact(in1 := "PCS_1".iCountReadR_fast, in2 := 9)
      I_Contact( "PCS_1".xREQR_fast )
      "PE_R_Module_4"(Input_Data := "PCS_1".arrDataR_fast, Output_Data => "PCS_1".R)
   END_RUNG
   // the same network as SCL:
   IF ("PCS_1".iCountReadR_fast = 9) AND NOT "PCS_1".xREQR_fast THEN
       "PE_R_Module_4"(Input_Data := "PCS_1".arrDataR_fast, Output_Data => "PCS_1".R);
   END_IF;
END_REGION

REGION Network 26: Write R_Block_10 parameter - Read Humidity module 1-2-3-4
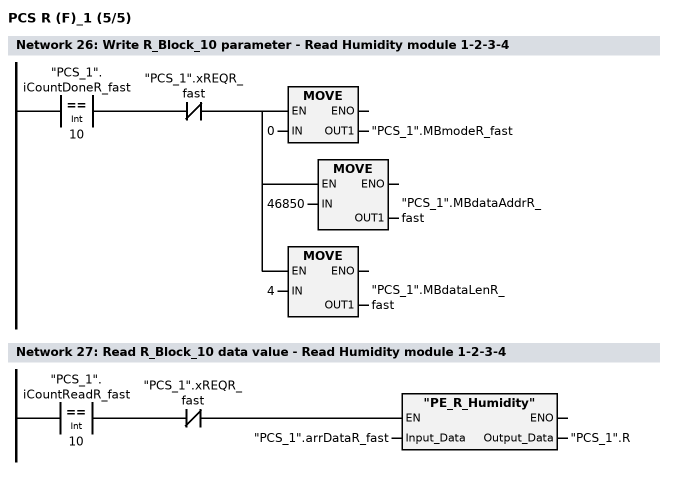
   RUNG wire#powerrail
      { S7_Templates := "SrcType := Int" } EQ_Contact(in1 := "PCS_1".iCountDoneR_fast, in2 := 10)
      I_Contact( "PCS_1".xREQR_fast )
      wire#w1
      Move(in := 0, out1 => "PCS_1".MBmodeR_fast)
   END_RUNG
   RUNG wire#w1
      Move(in := 46850, out1 => "PCS_1".MBdataAddrR_fast)
   END_RUNG
   RUNG wire#w1
      Move(in := 4, out1 => "PCS_1".MBdataLenR_fast)
   END_RUNG
   // the same network as SCL:
   IF ("PCS_1".iCountDoneR_fast = 10) AND NOT "PCS_1".xREQR_fast THEN
       "PCS_1".MBmodeR_fast := 0;
       "PCS_1".MBdataAddrR_fast := 46850;
       "PCS_1".MBdataLenR_fast := 4;
   END_IF;
END_REGION

REGION Network 27: Read R_Block_10 data value - Read Humidity module 1-2-3-4
   RUNG wire#powerrail
      { S7_Templates := "SrcType := Int" } EQ_Contact(in1 := "PCS_1".iCountReadR_fast, in2 := 10)
      I_Contact( "PCS_1".xREQR_fast )
      "PE_R_Humidity"(Input_Data := "PCS_1".arrDataR_fast, Output_Data => "PCS_1".R)
   END_RUNG
   // the same network as SCL:
   IF ("PCS_1".iCountReadR_fast = 10) AND NOT "PCS_1".xREQR_fast THEN
       "PE_R_Humidity"(Input_Data := "PCS_1".arrDataR_fast, Output_Data => "PCS_1".R);
   END_IF;
END_REGION
END_FUNCTION

FUNCTION "PCS W (F)_1" : Void   // FC48, LAD
TITLE = ModBus TCP for PCS Power Electronics
{ S7_Optimized_Access := 'TRUE' }
VERSION : 0.1
// stored: AutoNumber true, IsIECCheckEnabled false, SetENOAutomatically false, UDAEnableTagReadback false
   VAR_TEMP
      rSS1PacRef : Real;
      rSS2PacRef : Real;
      rSS1QacRef : Real;
      rSS2QacRef : Real;
      rSnHalfPE : Real;
      rQacRef : Real;
      uiQacRef : UInt;
   END_VAR
   VAR_TEMP   // added for the SCL form of the ladder/FBD networks
      _w1 : Bool;
   END_VAR
BEGIN

REGION Network 1: Function Modbus Client
